//
refGorn.xPowerOnFeedback:=xPowerOnFeedback;
refGorn.xInterlock:=xInterlock;
refGorn.xPowerEnable:= refGornRegisters.Read.strPowerSupplyControlRegister.sValue.COIL_VALUE[0];

{region "Blocked"}
IF refGorn.xInterlock  THEN
	refGorn.xBlocked:=TRUE;
ELSE
	refGorn.xBlocked:=FALSE;
END_IF
{endregion}
	 
{region "Setpoint check"}
refGorn.xAutoMode:=refGornSetting.xAutoMode;
refGorn.xModbusConnected:=xModbusConnected;	 
IF refGornSetting.xAutoMode THEN	 
	SpCurrent:=LIMIT(refGornSetting.rMinSpCurrent,refGornSetting.rAutoModeCurrent , refGornSetting.rMaxSpCurrent);
ELSE
	SpCurrent:=LIMIT(refGornSetting.rMinSpCurrent,refGornSetting.rSpCurrent , refGornSetting.rMaxSpCurrent); 
END_IF;
SpVoltage:=LIMIT(refGornSetting.rMinSpVoltage, refGornSetting.rSpVoltage , refGornSetting.rMaxSpVoltage);
{endregion}

refGorn.rSpCurrentFeedback :=refGornRegisters.Read.strSpCurrent.sValue.INT_VALUE;
										

refGorn.rSpVoltageFeedback := refGornRegisters.Read.strSpVoltage.sValue.INT_VALUE;
IF xCommand AND refGorn.xPowerEnable THEN
	refGorn.rFbCurrent := refGornRegisters.Read.strFbCurrent.sValue.INT_VALUE;
								
	refGorn.rFbVoltage := refGornRegisters.Read.strFbVolatge.sValue.INT_VALUE;						
ELSE
	refGorn.rFbCurrent := 0 ;
	refGorn.rFbVoltage := 0;
END_IF
{endregion}
	 
{region "Command"}
IF refGornSetting.xAutoMode AND NOT refGorn.xBlocked THEN
		refGorn.xManualCommand:=refGorn.xAutoCommand;
		refGorn.xManualPowerCommand:=refGorn.xAutoPowerCommand;
		
			
		xCommand:=refgorn.xAutoCommand;	 
END_IF
	 
IF NOT refGornSetting.xAutoMode AND NOT refGorn.xBlocked THEN
		refGorn.xAutoCommand:=refGorn.xManualCommand;
		refGorn.xAutoPowerCommand:=refGorn.xManualPowerCommand;
		
		xCommand:=refgorn.xManualCommand;	 
END_IF
	//OR refGorn.xStabVoltageError
IF  refGorn.xInternalError  OR refGorn.xStabCurrentError OR refGorn.xPowerError OR refGorn.xHeatProtect THEN
	refGorn.xAutoCommand:=			FALSE;
	
	refGorn.xManualCommand:= 		FALSE;


	xCommand:=						FALSE;
	refGorn.xError:=				TRUE;
	 
END_IF

IF refGorn.xBlocked THEN
	refGorn.xAutoCommand:=			FALSE;
	
	refGorn.xManualCommand:= 		FALSE;


	xCommand:=						FALSE;
END_IF
{endregion}

{region "CommandCoil"}

refGornRegisters.Write.strPowerSupplyControlRegister.sValue.COIL_VALUE[0]:=refGorn.xAutoPowerCommand OR refGorn.xManualPowerCommand ;
refGornRegisters.Write.strPowerSupplyControlRegister.sValue.COIL_VALUE[1]:=xCommand;
{endregion}
refGornRegisters.Write.strSpCurrent.sValue.INT_VALUE:=SpCurrent;
refGornRegisters.Write.strSpVoltage.sValue.INT_VALUE:=SpVoltage;	 
{region "ErrorStatus"}
IF refGornRegisters.Read.strPowerSupplyStatusRegister.sValue.COIL_VALUE[0] THEN
	refGorn.xInternalError:=TRUE;	 
END_IF
IF refGornRegisters.Read.strPowerSupplyStatusRegister.sValue.COIL_VALUE[1] THEN
	refGorn.xStabVoltageError:=TRUE;		 
END_IF
IF refGornRegisters.Read.strPowerSupplyStatusRegister.sValue.COIL_VALUE[2] THEN
	refGorn.xStabCurrentError:=TRUE;	 
END_IF
IF refGornRegisters.Read.strPowerSupplyStatusRegister.sValue.COIL_VALUE[3] THEN
	refGorn.xPowerError:= TRUE;	 
END_IF
IF refGornRegisters.Read.strPowerSupplyStatusRegister.sValue.COIL_VALUE[4] THEN
	refGorn.xHeatProtect:=TRUE;	 
END_IF
	 

IF xCommand AND refGorn.xPowerEnable AND refGorn.rFbCurrent>0.0 AND refGorn.rFbVoltage>0.0 THEN
	refGorn.xTurnOn:=TRUE;
ELSE
	refGorn.xTurnOn:=FALSE;		 
END_IF
		  
			   
IF refGorn.xAcknowledge THEN
	refGorn.xAcknowledge:=FALSE;
	refGorn.xInternalError:=FALSE;
 	refGorn.xStabVoltageError:=FALSE;
	refGorn.xStabCurrentError:=FALSE;
	refGorn.xPowerError:= FALSE;
	refGorn.xHeatProtect:=FALSE;		
	refGorn.xError:=FALSE; 
END_IF
{endregion}


	 


{region "output"}
xInternalError:=refGorn.xInternalError;
xStabVoltageError:=refGorn.xStabVoltageError;
xStabCurrentError:=refGorn.xStabCurrentError;
xPowerError:=refGorn.xPowerError;
xHeatProtect:=refGorn.xHeatProtect;
xRemoteStatus:=refGorn.xRemoteStatus;
xError:=refGorn.xError;
{endregion}

END_FUNCTION_BLOCK

// Function Blocks/Heater/fbHeater
FUNCTION_BLOCK fbHeater
VAR_INPUT
	Heater: 	REFERENCE TO udtHeater;
	Setting:	REFERENCE TO udtHeaterSetting;
	xInterlock:	BOOL;
	Temperature: REAL;
	TransIsOn:BOOL;
END_VAR
VAR_OUTPUT
	Power: UDINT;
	Command:BOOL;
END_VAR
VAR
	Regulator: Util.PID;
	LimitsActive:BOOL;
	Overflow:BOOL;
	SetPoint: REAL:=0;
END_VAR

Setting.rManualPower:=LIMIT(Setting.rMinPower, Setting.rManualPower, Setting.rMaxPower);
Heater.xPowerOn:=TransIsOn;
Heater.xLock := xInterlock;
Heater.Temepature:=THIS^.Temperature;

Heater.xError:= NOT Heater.xPowerOn OR Overflow;
SetPoint:=Setting.rSetpointTemperature;

IF Heater.xError OR Heater.xLock THEN
	SetPoint:=0;
	Heater.xManualCommand:=FALSE;
	Heater.xAutoCommand:=FALSE;
	
END_IF
IF  NOT Heater.xCommand THEN
	SetPoint:=0;
END_IF

Regulator(	ACTUAL:=Heater.Temepature,
			SET_POINT:=SetPoint,
			KP:= Setting.P,
			TN:= Setting.I,
			TV:= Setting.D,
			Y_Manual:=Setting.rManualPower*100,
			Y_OFFSET:=0,
			Y_MIN:=0.0,
			Y_MAX:=Setting.rMaxPower*100,
			MANUAL:= Setting.xManualPower,
			RESET:=Heater.xReset,
			Y=>Heater.rPower,
			LIMITS_ACTIVE=>LimitsActive,
			OVERFLOW=>Overflow);


	
IF NOT Setting.xAutoMode THEN
	Heater.xCommand:=Heater.xManualCommand;
	Heater.xAutoCommand:=Heater.xManualCommand;
ELSE
	Heater.xCommand:=Heater.xAutoCommand;
	Heater.xManualCommand:=Heater.xAutoCommand;
END_IF
 
IF Heater.xError THEN
	Heater.wState:=2;
ELSIF Heater.xLock THEN
	Heater.wState:=3;
ELSIF Heater.xCommand THEN
	Heater.wState:=1;
ELSE
	Heater.wState:=0;
END_IF

Command:=Heater.xCommand;
Power:=REAL_TO_UDINT(Heater.rPower);

END_FUNCTION_BLOCK

// Function Blocks/Inficon/fbInficon
FUNCTION_BLOCK fbInficon
VAR_INPUT
	Inficon:			REFERENCE TO udtInficon;
	SendSize:  			REFERENCE TO UINT;
	pSendBuffer:		POINTER TO BYTE; //Указатель на массив отправки сообщения
	iSendBufferLength: 	INT;
	pRcvBuffer:			POINTER TO BYTE;
	pRcvSize:			INT; //Количество полученных байт;
	xSendMessageReady:	REFERENCE TO BOOL;//Сигнал о готовности сообщения для отправки
	xRcvFlagDone:		BOOL; //Флаг о завершение принятия данных
	pMessageBuffer: 	POINTER TO BYTE; //Указатель на байтовый массив, который будет использоваться как буффер для составления Message
	iMessageBuffferLength: INT;//Длина массива, который используется как буффер
	COMPortIsOpened:	BOOL;
	
	InficonResponce: POINTER TO udtInficonResponcePackage;
	
	InficonRemoteGeneralActionResponce: POINTER TO udtRemoteGeneralActionResponce;
END_VAR
VAR_OUTPUT
END_VAR
VAR
	MessageBuffer:		fbGeneralBuffer;//Функциональный блок для работы с буффером
	SendBuffer:			fbGeneralBuffer;
	
	Query: 				fbInficonQuery;
	Update: 			fbInficonUpdate;
	Status:				fbInficonStatus;
	Remote:				fbInficonRemote;
	STAGE: 				INT;
	xMesaageBufferEmpty:BOOL;
	xMessageBufferInit: BOOL:=FALSE;
	xSendBufferEmpty:	BOOL;
	HelloComadResult: 	INT;

	RawMessageLength: 	DINT;
	BufferPointer: 		POINTER TO ARRAY[0..1] OF BYTE;
	
	SensoreStatusResult:INT; //Реультат выполнения стадии опроса сенсоров
	CRCResult: 			BYTE;
	
	SensoreStatusStage: INT; //Этапы выполнения стадии опроса сенсоров
	RemoteGeneralActionResult: 	INT; //Результат выполнения стадии команд
	RemoteGeneralActionStage:	INT;
	
	getFiltredRateStage: INT;
	getFiltredRateRsult: INT;
	InficonResponceSMFilteredRate: udtInficonResponceSMFiltredrate;
	
	
	
END_VAR

IF NOT xMessageBufferInit THEN
	MessageBuffer(pBuffer:=pMessageBuffer,
			pBufferLength:=iMessageBuffferLength,
			xEmpty=>xMesaageBufferEmpty,
			xInit=>xMessageBufferInit);
	SendBuffer(	pBuffer:=pSendBuffer,
				pBufferLength:=iSendBufferLength,
				xEmpty=>xSendBufferEmpty,
				xInit=>xMessageBufferInit);
	THIS^.Status(MessageBuffer:=ADR(MessageBuffer));
	THIS^.Remote(MessageBuffer:=ADR(MessageBuffer));
	BufferPointer:=ADR(RawMessageLength);		
END_IF




CASE STAGE OF
	InficonStage.WAIT:
		IF COMPortIsOpened THEN
			STAGE:=InficonStage.STATUS_SENSORE;
		END_IF
		
	InficonStage.STATUS_SENSORE:
		SensoreStatusResult:=THIS^.SensoreStatus(SensoreStatusStage);
		IF SensoreStatusResult = InficonMethodStatus.COMPLETE THEN
			Stage:=InficonStage.GET_MATERIAL_FILTRED_RATE;
		END_IF
		IF SensoreStatusResult = InficonMethodStatus.ERROR THEN
			Stage:= InficonStage.ERROR;
		END_IF
	InficonStage.GET_MATERIAL_FILTRED_RATE:
		getFiltredRateRsult :=THIS^.GetMateriaFiltredRate(Stage:=getFiltredRateStage);
		IF getFiltredRateRsult = InficonMethodStatus.COMPLETE THEN
			Stage:=InficonStage.REMOTE_GENERAL_ACTION;
		END_IF
		IF getFiltredRateRsult = InficonMethodStatus.ERROR THEN
			Stage:= InficonStage.ERROR;
		END_IF		
	InficonStage.REMOTE_GENERAL_ACTION:
		IF Inficon.xManualReset_1 THEN
			RemoteGeneralActionResult:=THIS^.RemoteGeneralAction(RemoteGeneralActionStage,16#01);
			IF RemoteGeneralActionResult = InficonMethodStatus.COMPLETE THEN
				Inficon.xManualReset_1:=FALSE;
				Stage:=InficonStage.WAIT;
			END_IF
			IF RemoteGeneralActionResult = InficonMethodStatus.ERROR THEN
				Stage:= InficonStage.ERROR;
			END_IF
		ELSIF Inficon.xManualReset_2 THEN
			RemoteGeneralActionResult:=THIS^.RemoteGeneralAction(RemoteGeneralActionStage,16#02);
			IF RemoteGeneralActionResult = InficonMethodStatus.COMPLETE THEN
				Inficon.xManualReset_2:=FALSE;
				Stage:=InficonStage.WAIT;
			END_IF
			IF RemoteGeneralActionResult = InficonMethodStatus.ERROR THEN
				Stage:= InficonStage.ERROR;
			END_IF
		ELSIF Inficon.xManualReset_3 THEN
			RemoteGeneralActionResult:=THIS^.RemoteGeneralAction(RemoteGeneralActionStage,16#03);
			IF RemoteGeneralActionResult = InficonMethodStatus.COMPLETE THEN
				Inficon.xManualReset_3:=FALSE;
				Stage:=InficonStage.WAIT;
			END_IF
			IF RemoteGeneralActionResult = InficonMethodStatus.ERROR THEN
				Stage:= InficonStage.ERROR;
			END_IF
		ELSIF
			Inficon.xManualReset_4 THEN
			RemoteGeneralActionResult:=THIS^.RemoteGeneralAction(RemoteGeneralActionStage,16#04);
			IF RemoteGeneralActionResult = InficonMethodStatus.COMPLETE THEN
				Inficon.xManualReset_4:=FALSE;
				Stage:=InficonStage.WAIT;
			END_IF
			IF RemoteGeneralActionResult = InficonMethodStatus.ERROR THEN
				Stage:= InficonStage.ERROR;
			END_IF
		ELSIF Inficon.xManualReset_5 THEN
			RemoteGeneralActionResult:=THIS^.RemoteGeneralAction(RemoteGeneralActionStage,16#05);
			IF RemoteGeneralActionResult = InficonMethodStatus.COMPLETE THEN
				Inficon.xManualReset_5:=FALSE;
				Stage:=InficonStage.WAIT;
			END_IF
			IF RemoteGeneralActionResult = InficonMethodStatus.ERROR THEN
				Stage:= InficonStage.ERROR;
			END_IF
		ELSIF Inficon.xManualReset_6 THEN
			RemoteGeneralActionResult:=THIS^.RemoteGeneralAction(RemoteGeneralActionStage,16#06);
			IF RemoteGeneralActionResult = InficonMethodStatus.COMPLETE THEN
				Inficon.xManualReset_6:=FALSE;
				Stage:=InficonStage.WAIT;
			END_IF
			IF RemoteGeneralActionResult = InficonMethodStatus.ERROR THEN
				Stage:= InficonStage.ERROR;
			END_IF
		ELSE
			Stage:=InficonStage.WAIT;
		END_IF
		

	InficonStage.ERROR:
		IF Inficon.xAcknowledge THEN
			Inficon.xAcknowledge:=FALSE;
			Stage:=InficonStage.WAIT;
		END_IF
	
// 	
// 	10:
// 		HelloComadResult:=THIS^.HelloCommand(16#01);
// 		IF HelloComadResult<>-1 THEN
// 			Stage:=11;
// 		END_IF
// 	11:
// 		RawMessageLength:=MessageBuffer.getBufferLength;
// 
// 		SendBuffer.AddElement(BufferPointer^[0]);
// 		SendBuffer.AddElement(BufferPointer^[1]);
// 		Stage:=12;
// 	12:
// 		SendBuffer.AddStruct(pData:=MessageBuffer.getBufferAddres,
// 							Length:=DINT_TO_INT(MessageBuffer.getBufferLength));
// 		Stage:=13;
// 	13:
// 		CRCResult:=THIS^.CalcCRC(Message:=SendBuffer.getBufferAddres,
// 									Length:=SendBuffer.getBufferLength);
// 		Stage:=14;
// 	14:
// 		SendBuffer.AddElement(THIS^.CRCResult);
// 		xSendMessageReady:=TRUE;
// 		Stage:=0;
// 		
		
END_CASE

METHOD ADD_Sensore : INT
VAR_INPUT
	SensoreNumber: BYTE;
END_VAR
END_METHOD

(*Расчет CRC*)
METHOD CalcCRC : BYTE
VAR_INPUT
	Message: POINTER TO BYTE;
	Length: DINT;
END_VAR
VAR
	Counter: DINT;
	InnerMessage: POINTER TO BYTE;
END_VAR
CalcCRC:=0;

FOR Counter:=0 TO Length-1 DO
	InnerMessage :=Message+Counter;
	CalcCRC:=CalcCRC+InnerMessage^;
END_FOR

CalcCRC:=CalcCRC AND 255;
END_METHOD

METHOD GetMateriaFiltredRate : INT
VAR_INPUT
	Stage: 					REFERENCE TO INT;
END_VAR
VAR
	AddCommandResult: 		INT;
	ClearMessageResult: 	INT; //Результат выполнения отчистки буффера сообщений
	ClearSendBufferResult:	INT; //Результат выполнения очистки буффера отправки
	RawLength: 				DINT;
	MessageLengthForBuffer: POINTER TO ARRAY[0..1] OF BYTE;
	CRCResult: 				BYTE;
	rTempFloat:				POINTER TO REAL;
END_VAR
CASE Stage OF
	InficonMethodStage.WAIT:
		GetMateriaFiltredRate:=InficonMethodState.BUSY;
		ClearMessageResult:=THIS^.MessageBuffer.ClearBuffer();
		ClearSendBufferResult:=THIS^.SendBuffer.ClearBuffer();
		IF ClearMessageResult = 200 AND ClearSendBufferResult = 200 THEN
			Stage:=InficonMethodStage.ADD_COMMAND;
		END_IF
	InficonMethodStage.ADD_COMMAND:
		AddCommandResult:=THIS^.Status.Material(CommandID:=InficonSLCommandID.FilteredRate, MaterialNumber:=16#0);
		IF AddCommandResult = -1THEN
			GetMateriaFiltredRate := InficonMethodState.ERROR;
			RETURN;
		END_IF
		Stage:=InficonMethodStage.ADD_LENGTH_TO_SENDBUFFER;
	InficonMethodStage.ADD_LENGTH_TO_SENDBUFFER:
		RawLength:=THIS^.MessageBuffer.getBufferLength;
		MessageLengthForBuffer:=ADR(RawLength);
		THIS^.SendBuffer.AddElement(pData:=MessageLengthForBuffer^[0]);
		THIS^.SendBuffer.AddElement(pData:=MessageLengthForBuffer^[1]);
		Stage:=InficonMethodStage.CALC_CRC;
	InficonMethodStage.CALC_CRC:
		CRCResult:=THIS^.CalcCRC(Message:=THIS^.MessageBuffer.getBufferAddres,
									Length:=THIS^.MessageBuffer.getBufferLength);
		THIS^.MessageBuffer.AddElement(pData:=CRCResult);
		Stage:=InficonMethodStage.ADD_CRC;
	InficonMethodStage.ADD_CRC:
		Stage:=InficonMethodStage.ADD_DATA_TO_SENDBUFFER;
	InficonMethodStage.ADD_DATA_TO_SENDBUFFER:
		THIS^.SendBuffer.AddStruct(pData:=THIS^.MessageBuffer.getBufferAddres,
								Length:=DINT_TO_INT(THIS^.MessageBuffer.getBufferLength));
		Stage:=InficonMethodStage.EDGE_MESSAGECOMPLETE_FLAG;		
	InficonMethodStage.EDGE_MESSAGECOMPLETE_FLAG:
		THIS^.SendSize:=DINT_TO_UINT(THIS^.SendBuffer.getBufferLength);
		THIS^.xSendMessageReady:=TRUE;
		Stage:=InficonMethodStage.WAIT_RESPONCE;
	InficonMethodStage.WAIT_RESPONCE:
		IF THIS^.xRcvFlagDone THEN
			Stage:=InficonMethodStage.PARSE_RESPONCE;
		END_IF
	InficonMethodStage.PARSE_RESPONCE:
		MEMUtils.MemCpy(pbyDest:=ADR(THIS^.InficonResponceSMFilteredRate),
						pbySrc:=pRcvBuffer,
						dwSize:=5);
		Stage:=InficonMethodStage.CHECK_RESPONCE_STATUS;		
	InficonMethodStage.CHECK_RESPONCE_STATUS:
		IF InficonResponceSMFilteredRate.Code<>16#6 THEN
			Stage:=InficonMethodStage.COMPLETE;
			RETURN;
		END_IF
		
		MEMUtils.MemCpy(pbyDest:=ADR(THIS^.InficonResponceSMFilteredRate),
						pbySrc:=pRcvBuffer,
						dwSize:=SIZEOF(udtInficonResponceSMFiltredrate));
						
		THIS^.Inficon.Materials.FilteredRate[0].vValue[0]:=InficonResponceSMFilteredRate.FR_1_1;
		THIS^.Inficon.Materials.FilteredRate[0].vValue[1]:=InficonResponceSMFilteredRate.FR_1_2;
		THIS^.Inficon.Materials.FilteredRate[0].vValue[2]:=InficonResponceSMFilteredRate.FR_1_3;
		THIS^.Inficon.Materials.FilteredRate[0].vValue[3]:=InficonResponceSMFilteredRate.FR_1_4;

		THIS^.Inficon.Materials.FilteredRate[1].vValue[0]:=InficonResponceSMFilteredRate.FR_2_1;
		THIS^.Inficon.Materials.FilteredRate[1].vValue[1]:=InficonResponceSMFilteredRate.FR_2_2;
		THIS^.Inficon.Materials.FilteredRate[1].vValue[2]:=InficonResponceSMFilteredRate.FR_2_3;
		THIS^.Inficon.Materials.FilteredRate[1].vValue[3]:=InficonResponceSMFilteredRate.FR_2_4;
		
		THIS^.Inficon.Materials.FilteredRate[2].vValue[0]:=InficonResponceSMFilteredRate.FR_3_1;
		THIS^.Inficon.Materials.FilteredRate[2].vValue[1]:=InficonResponceSMFilteredRate.FR_3_2;
		THIS^.Inficon.Materials.FilteredRate[2].vValue[2]:=InficonResponceSMFilteredRate.FR_3_3;
		THIS^.Inficon.Materials.FilteredRate[2].vValue[3]:=InficonResponceSMFilteredRate.FR_3_4;

		THIS^.Inficon.Materials.FilteredRate[3].vValue[0]:=InficonResponceSMFilteredRate.FR_4_1;
		THIS^.Inficon.Materials.FilteredRate[3].vValue[1]:=InficonResponceSMFilteredRate.FR_4_2;
		THIS^.Inficon.Materials.FilteredRate[3].vValue[2]:=InficonResponceSMFilteredRate.FR_4_3;
		THIS^.Inficon.Materials.FilteredRate[3].vValue[3]:=InficonResponceSMFilteredRate.FR_4_4;

		THIS^.Inficon.Materials.FilteredRate[4].vValue[0]:=InficonResponceSMFilteredRate.FR_5_1;
		THIS^.Inficon.Materials.FilteredRate[4].vValue[1]:=InficonResponceSMFilteredRate.FR_5_2;
		THIS^.Inficon.Materials.FilteredRate[4].vValue[2]:=InficonResponceSMFilteredRate.FR_5_3;
		THIS^.Inficon.Materials.FilteredRate[4].vValue[3]:=InficonResponceSMFilteredRate.FR_5_4;

		THIS^.Inficon.Materials.FilteredRate[5].vValue[0]:=InficonResponceSMFilteredRate.FR_6_1;
		THIS^.Inficon.Materials.FilteredRate[5].vValue[1]:=InficonResponceSMFilteredRate.FR_6_2;
		THIS^.Inficon.Materials.FilteredRate[5].vValue[2]:=InficonResponceSMFilteredRate.FR_6_3;
		THIS^.Inficon.Materials.FilteredRate[5].vValue[3]:=InficonResponceSMFilteredRate.FR_6_4;
		
		Stage:=InficonMethodStage.COMPLETE;
	InficonMethodStage.COMPLETE:
		Stage:=InficonMethodStage.WAIT;
		GetMateriaFiltredRate:=InficonMethodStatus.COMPLETE;
	InficonMethodStage.ERROR:
	
	
	
END_CASE
END_METHOD

METHOD HCPub : INT
VAR_INPUT
	CommandID:BYTE;
END_VAR
HCPub:=HelloCommand(CommandID:=CommandID);
END_METHOD

(*
HelloComand - метод формируюзий Hello Command запрос
Формат запроса: H<CommandID>
*)
METHOD PROTECTED HelloCommand : INT
VAR_INPUT
	CommandID:BYTE;
END_VAR
VAR
	CRC:BYTE;
END_VAR
THIS^.MessageBuffer.ClearBuffer();
HelloCommand:=THIS^.MessageBuffer.AddElement(pData:=InficonCommand.Hello,
							);
IF HelloCommand = -1 THEN
	RETURN;
END_IF
	
HelloCommand:=THIS^.MessageBuffer.AddElement(pData:=CommandID,
							);

			
IF HelloCommand = -1 THEN
	RETURN;
END_IF
END_METHOD

METHOD RemoteGeneralAction : INT
VAR_INPUT
	Stage: REFERENCE TO INT;
	MaterialNumber: BYTE;
	
END_VAR
VAR
	ClearMessageResult: 	INT; //Результат выполнения отчистки буффера сообщений
	ClearSendBufferResult:	INT; //Результат выполнения очистки буффера отправки
	AddCommandResult: 		INT;
	RawLength: 				DINT; //Длина сообщения
	MessageLengthForBuffer: POINTER TO ARRAY[0..1] OF BYTE;
	CRCResult: 				BYTE; 
	
	
END_VAR
CASE Stage OF
	

	InficonMethodStage.WAIT:
		RemoteGeneralAction:=InficonMethodState.BUSY;
		ClearMessageResult:=THIS^.MessageBuffer.ClearBuffer();
		ClearSendBufferResult:=THIS^.SendBuffer.ClearBuffer();
		IF ClearMessageResult = 200 AND ClearSendBufferResult = 200 THEN
			Stage:=InficonMethodStage.ADD_COMMAND;
		END_IF
	
		
	InficonMethodStage.ADD_COMMAND:
		AddCommandResult:=THIS^.Remote.MaterialAction(CommandID:=InficonRLCommandID.ZeroThickness,
													MaterialNumber:=MaterialNumber,
													pData:=0,
													Length:=0);
		IF AddCommandResult= -1 THEN
			RemoteGeneralAction:=InficonMethodState.ERROR;
			RETURN;
		END_IF
		Stage:=InficonMethodStage.ADD_LENGTH_TO_SENDBUFFER;
	
		
	InficonMethodStage.ADD_LENGTH_TO_SENDBUFFER:
		RawLength:=THIS^.MessageBuffer.getBufferLength;
		MessageLengthForBuffer:=ADR(RawLength);
		THIS^.SendBuffer.AddElement(pData:=MessageLengthForBuffer^[0]);
		THIS^.SendBuffer.AddElement(pData:=MessageLengthForBuffer^[1]);
		Stage:=InficonMethodStage.CALC_CRC;
		
		
	InficonMethodStage.CALC_CRC:
		CRCResult:=THIS^.CalcCRC(Message:=THIS^.MessageBuffer.getBufferAddres,
									Length:=THIS^.MessageBuffer.getBufferLength);
		THIS^.MessageBuffer.AddElement(pData:=CRCResult);
		Stage:=InficonMethodStage.ADD_DATA_TO_SENDBUFFER;
		
		
	InficonMethodStage.ADD_DATA_TO_SENDBUFFER:
		THIS^.SendBuffer.AddStruct(pData:=THIS^.MessageBuffer.getBufferAddres,
								Length:=DINT_TO_INT(THIS^.MessageBuffer.getBufferLength));
		Stage:=InficonMethodStage.EDGE_MESSAGECOMPLETE_FLAG;
		
		
	InficonMethodStage.EDGE_MESSAGECOMPLETE_FLAG:
		THIS^.SendSize:=DINT_TO_UINT(THIS^.SendBuffer.getBufferLength);
		THIS^.xSendMessageReady:=TRUE;
		Stage:=InficonMethodStage.WAIT_RESPONCE;
	
		
	InficonMethodStage.WAIT_RESPONCE:
		IF THIS^.xRcvFlagDone THEN
			Stage:=InficonMethodStage.PARSE_RESPONCE;
		END_IF
	
		
	InficonMethodStage.PARSE_RESPONCE:
		MEMUtils.MemCpy(pbyDest:=THIS^.InficonRemoteGeneralActionResponce,
						pbySrc:=pRcvBuffer,
						dwSize:=THIS^.pRcvSize);
		Stage:=InficonMethodStage.CHECK_RESPONCE_STATUS;
	
		
	InficonMethodStage.CHECK_RESPONCE_STATUS:
	
			Stage:=InficonMethodStage.COMPLETE;

		THIS^.xSendMessageReady:=FALSE;
		THIS^.xRcvFlagDone:=TRUE;
		
		
	InficonMethodStage.COMPLETE:
		Stage:=InficonMethodStage.WAIT;
		RemoteGeneralAction:=InficonMethodStatus.COMPLETE;
		
	InficonMethodStage.ERROR:
END_CASE
END_METHOD

METHOD SensoreStatus : INT
VAR_INPUT
	Stage: REFERENCE TO INT;
END_VAR
VAR
	AddCommandResult: INT;
	ClearMessageResult: INT; //Результат выполнения отчистки буффера сообщений
	ClearSendBufferResult:INT; //Результат выполнения очистки буффера отправки
	RawLength: DINT;
	MessageLengthForBuffer: POINTER TO ARRAY[0..1] OF BYTE;
	CRCResult: BYTE;
	rTempFloat:POINTER TO REAL;
	
END_VAR
CASE Stage OF
	InficonMethodStage.WAIT:
	
		//Инициализация массивов
		SensoreStatus:=InficonMethodState.BUSY;
		ClearMessageResult:=THIS^.MessageBuffer.ClearBuffer();
		ClearSendBufferResult:=THIS^.SendBuffer.ClearBuffer();
		IF ClearMessageResult = 200 AND ClearSendBufferResult = 200 THEN
			Stage:=InficonMethodStage.ADD_COMMAND;
		END_IF
		
	InficonMethodStage.ADD_COMMAND:
		//Запись команды получения значения всех скоростей напыления
		AddCommandResult:=THIS^.Status.Sensor(CommandID:=InficonSSCommandID.SensorThickness, SensorNumber:=16#0);
		IF AddCommandResult= -1 THEN
			SensoreStatus:=InficonMethodState.ERROR;
			RETURN;
		END_IF
		Stage:=InficonMethodStage.ADD_LENGTH_TO_SENDBUFFER;

	InficonMethodStage.ADD_LENGTH_TO_SENDBUFFER:
	
		RawLength:=THIS^.MessageBuffer.getBufferLength;
		MessageLengthForBuffer:=ADR(RawLength);
		THIS^.SendBuffer.AddElement(pData:=MessageLengthForBuffer^[0]);
		THIS^.SendBuffer.AddElement(pData:=MessageLengthForBuffer^[1]);
		Stage:=InficonMethodStage.CALC_CRC;
	
	InficonMethodStage.CALC_CRC:
		
		CRCResult:=THIS^.CalcCRC(Message:=THIS^.MessageBuffer.getBufferAddres,
									Length:=THIS^.MessageBuffer.getBufferLength);
		THIS^.MessageBuffer.AddElement(pData:=CRCResult);
		Stage:=InficonMethodStage.ADD_CRC;
		
	InficonMethodStage.ADD_CRC:
		Stage:=InficonMethodStage.ADD_DATA_TO_SENDBUFFER;
		
	InficonMethodStage.ADD_DATA_TO_SENDBUFFER:
		THIS^.SendBuffer.AddStruct(pData:=THIS^.MessageBuffer.getBufferAddres,
								Length:=DINT_TO_INT(THIS^.MessageBuffer.getBufferLength));
		Stage:=InficonMethodStage.EDGE_MESSAGECOMPLETE_FLAG;
		
	InficonMethodStage.EDGE_MESSAGECOMPLETE_FLAG:
		THIS^.SendSize:=DINT_TO_UINT(THIS^.SendBuffer.getBufferLength);
		THIS^.xSendMessageReady:=TRUE;
		Stage:=InficonMethodStage.WAIT_RESPONCE;
		
	InficonMethodStage.WAIT_RESPONCE:
		IF THIS^.xRcvFlagDone THEN
			Stage:=InficonMethodStage.PARSE_RESPONCE;
		END_IF
	InficonMethodStage.PARSE_RESPONCE:
		MEMUtils.MemCpy(pbyDest:=InficonResponce,
						pbySrc:=pRcvBuffer,
						dwSize:=5);
		Stage:=InficonMethodStage.CHECK_RESPONCE_STATUS;
		
	InficonMethodStage.CHECK_RESPONCE_STATUS:
		IF InficonResponce^.Code<>16#6 THEN
			Stage:=InficonMethodStage.COMPLETE;
			RETURN;
		END_IF
		
		MEMUtils.MemCpy(pbyDest:=InficonResponce,
						pbySrc:=pRcvBuffer,
						dwSize:=SIZEOF(udtInficonResponcePackage));
						
		(*MEMUtils.SwapLocalToMotorola(pAddress:=ADR(InficonResponce^.Thinkness_1_1),
								iSize:=4);
		rTempFloat:= ADR(InficonResponce^.Thinkness_1_1);
		THIS^.Inficon.Sensore1Thickness:=rTempFloat^;*)
		THIS^.Inficon.Sensore1Thickness.vValue[0]:=InficonResponce^.Thinkness_1_1;
		THIS^.Inficon.Sensore1Thickness.vValue[1]:=InficonResponce^.Thinkness_1_2;
		THIS^.Inficon.Sensore1Thickness.vValue[2]:=InficonResponce^.Thinkness_1_3;
		THIS^.Inficon.Sensore1Thickness.vValue[3]:=InficonResponce^.Thinkness_1_4;

		THIS^.Inficon.Sensore2Thickness.vValue[0]:=InficonResponce^.Thinkness_2_1;
		THIS^.Inficon.Sensore2Thickness.vValue[1]:=InficonResponce^.Thinkness_2_2;
		THIS^.Inficon.Sensore2Thickness.vValue[2]:=InficonResponce^.Thinkness_2_3;
		THIS^.Inficon.Sensore2Thickness.vValue[3]:=InficonResponce^.Thinkness_2_4;
		
		THIS^.Inficon.Sensore3Thickness.vValue[0]:=InficonResponce^.Thinkness_3_1;
		THIS^.Inficon.Sensore3Thickness.vValue[1]:=InficonResponce^.Thinkness_3_2;
		THIS^.Inficon.Sensore3Thickness.vValue[2]:=InficonResponce^.Thinkness_3_3;
		THIS^.Inficon.Sensore3Thickness.vValue[3]:=InficonResponce^.Thinkness_3_4;

		THIS^.Inficon.Sensore4Thickness.vValue[0]:=InficonResponce^.Thinkness_4_1;
		THIS^.Inficon.Sensore4Thickness.vValue[1]:=InficonResponce^.Thinkness_4_2;
		THIS^.Inficon.Sensore4Thickness.vValue[2]:=InficonResponce^.Thinkness_4_3;
		THIS^.Inficon.Sensore4Thickness.vValue[3]:=InficonResponce^.Thinkness_4_4;

		THIS^.Inficon.Sensore5Thickness.vValue[0]:=InficonResponce^.Thinkness_5_1;
		THIS^.Inficon.Sensore5Thickness.vValue[1]:=InficonResponce^.Thinkness_5_2;
		THIS^.Inficon.Sensore5Thickness.vValue[2]:=InficonResponce^.Thinkness_5_3;
		THIS^.Inficon.Sensore5Thickness.vValue[3]:=InficonResponce^.Thinkness_5_4;

		THIS^.Inficon.Sensore6Thickness.vValue[0]:=InficonResponce^.Thinkness_6_1;
		THIS^.Inficon.Sensore6Thickness.vValue[1]:=InficonResponce^.Thinkness_6_2;
		THIS^.Inficon.Sensore6Thickness.vValue[2]:=InficonResponce^.Thinkness_6_3;
		THIS^.Inficon.Sensore6Thickness.vValue[3]:=InficonResponce^.Thinkness_6_4;
		Stage:=InficonMethodStage.COMPLETE;
		
		
		
		
	InficonMethodStage.COMPLETE:
		Stage:=InficonMethodStage.WAIT;
		SensoreStatus:=InficonMethodStatus.COMPLETE;
	InficonMethodStage.ERROR:
END_CASE
END_METHOD

END_FUNCTION_BLOCK

// Function Blocks/Inficon/fbInficonQuery
FUNCTION_BLOCK fbInficonQuery
VAR_INPUT
	MessageBuffer: POINTER TO fbGeneralBuffer;
END_VAR
VAR_OUTPUT
END_VAR
VAR
END_VAR

THIS^.MessageBuffer^.ClearBuffer();
THIS^.MessageBuffer^.AddElement(pData:=InficonCommand.Query,);

(*
QG<CommandID>
*)
METHOD PUBLIC General : INT
VAR_INPUT
	CommandID:BYTE;
END_VAR
THIS^();

General:=THIS^.MessageBuffer^.AddElement(pData:=InficonQUSubgroup.General);
IF General = -1 THEN
	RETURN;
END_IF

General:=THIS^.MessageBuffer^.AddElement(pData:=CommandID);	
IF General = -1 THEN
	RETURN;
END_IF
END_METHOD

METHOD PUBLIC Material : INT
VAR_INPUT
	CommandID: BYTE;
	MaterialNumber:BYTE;
END_VAR
THIS^();

Material:= THIS^.MessageBuffer^.AddElement(pData:=InficonQUSubgroup.Material);
IF Material = -1 THEN
	RETURN;
END_IF

Material:= THIS^.MessageBuffer^.AddElement(pData:=CommandID);
IF Material = -1 THEN
	RETURN;
END_IF

Material:= THIS^.MessageBuffer^.AddElement(pData:=MaterialNumber);
IF Material = -1 THEN
	RETURN;
END_IF
END_METHOD

METHOD PUBLIC ProcessMaterial : INT
VAR_INPUT
	CommandID: BYTE;
	ProcessNumber:BYTE;
	MaterialNumber:BYTE;
END_VAR
THIS^();



ProcessMaterial:= THIS^.MessageBuffer^.AddElement(pData:=InficonQUSubgroup.Process);
IF ProcessMaterial = -1 THEN
	RETURN;
END_IF



ProcessMaterial:= THIS^.MessageBuffer^.AddElement(pData:=CommandID);
IF ProcessMaterial = -1 THEN
	RETURN;
END_IF

ProcessMaterial:= THIS^.MessageBuffer^.AddElement(pData:=ProcessNumber);
IF ProcessMaterial = -1 THEN
	RETURN;
END_IF

ProcessMaterial:= THIS^.MessageBuffer^.AddElement(pData:=MaterialNumber);
IF ProcessMaterial = -1 THEN
	RETURN;
END_IF
END_METHOD

METHOD PUBLIC Sensor : INT
VAR_INPUT
	CommandID: BYTE;
	SensorNumber:BYTE;
END_VAR
THIS^();

Sensor:= THIS^.MessageBuffer^.AddElement(pData:=InficonQUSubgroup.Sensor);
IF Sensor = -1 THEN
	RETURN;
END_IF

Sensor:= THIS^.MessageBuffer^.AddElement(pData:=CommandID);
IF Sensor = -1 THEN
	RETURN;
END_IF

Sensor:= THIS^.MessageBuffer^.AddElement(pData:=SensorNumber);
IF Sensor = -1 THEN
	RETURN;
END_IF
END_METHOD

METHOD PUBLIC Source : INT
VAR_INPUT	
	CommandID: BYTE;
	SourceNumber:BYTE;
END_VAR
THIS^();

Source:= THIS^.MessageBuffer^.AddElement(pData:=InficonQUSubgroup.Source);
IF Source = -1 THEN
	RETURN;
END_IF

Source:= THIS^.MessageBuffer^.AddElement(pData:=CommandID);
IF Source = -1 THEN
	RETURN;
END_IF

Source:= THIS^.MessageBuffer^.AddElement(pData:=SourceNumber);
IF Source = -1 THEN
	RETURN;
END_IF
END_METHOD

END_FUNCTION_BLOCK

// Function Blocks/Inficon/fbInficonUpdate
FUNCTION_BLOCK fbInficonUpdate
VAR_INPUT
	MessageBuffer: POINTER TO fbGeneralBuffer;
END_VAR
VAR_OUTPUT
END_VAR
VAR
END_VAR

THIS^.MessageBuffer^.ClearBuffer();
THIS^.MessageBuffer^.AddElement(pData:=InficonCommand.Update);

METHOD PUBLIC General : INT
VAR_INPUT
	CommandID:BYTE;
	pData: POINTER TO BYTE;
	Length:INT;
END_VAR
THIS^();

General := THIS^.MessageBuffer^.AddElement(pData:=InficonQUSubgroup.General);
IF General = -1 THEN
	RETURN;
END_IF

General:=THIS^.MessageBuffer^.AddElement(pData:=CommandID);
IF General= -1 THEN
	RETURN;
END_IF

General:=THIS^.MessageBuffer^.AddStruct(pData:=pData,
			Length:=Length);
IF General = -1 THEN
	RETURN;
END_IF
END_METHOD

METHOD PUBLIC Material : INT
VAR_INPUT
	CommandID: BYTE;
	MaterialNumber:BYTE;
	pData: POINTER TO BYTE;
	Length:INT;
END_VAR
THIS^();

Material:= THIS^.MessageBuffer^.AddElement(pData:=InficonQUSubgroup.Material);
IF Material = -1 THEN
	RETURN;
END_IF

Material:= THIS^.MessageBuffer^.AddElement(pData:=CommandID);
IF Material = -1 THEN
	RETURN;
END_IF

Material:= THIS^.MessageBuffer^.AddElement(pData:=MaterialNumber);
IF Material = -1 THEN
	RETURN;
END_IF

Material:=THIS^.MessageBuffer^.AddStruct(pData:=pData,
	Length:=Length);
IF Material = -1 THEN
	RETURN;
END_IF
END_METHOD

METHOD PUBLIC ProcessMaterial : INT
VAR_INPUT
	CommandID: BYTE;
	ProcessNumber:BYTE;
	MaterialNumber:BYTE;
	pData: POINTER TO BYTE;
	Length:INT;
END_VAR
THIS^();

ProcessMaterial:= THIS^.MessageBuffer^.AddElement(pData:=InficonQUSubgroup.Process);
IF ProcessMaterial = -1 THEN
	RETURN;
END_IF

ProcessMaterial:= THIS^.MessageBuffer^.AddElement(pData:=CommandID);
IF ProcessMaterial = -1 THEN
	RETURN;
END_IF

ProcessMaterial:= THIS^.MessageBuffer^.AddElement(pData:=ProcessNumber);
IF ProcessMaterial = -1 THEN
	RETURN;
END_IF

ProcessMaterial:= THIS^.MessageBuffer^.AddElement(pData:=MaterialNumber);
IF ProcessMaterial = -1 THEN
	RETURN;
END_IF

ProcessMaterial:=THIS^.MessageBuffer^.AddStruct(pData:=pData,
	Length:=Length);
IF ProcessMaterial = -1 THEN
	RETURN;
END_IF
END_METHOD

METHOD PUBLIC Sensor : INT
VAR_INPUT
	CommandID: BYTE;
	SensorNumber:BYTE;
	pData: POINTER TO BYTE;
	Length:INT;
END_VAR
THIS^();

Sensor:= THIS^.MessageBuffer^.AddElement(pData:=InficonQUSubgroup.Sensor);
IF Sensor = -1 THEN
	RETURN;
END_IF

Sensor:= THIS^.MessageBuffer^.AddElement(pData:=CommandID);
IF Sensor = -1 THEN
	RETURN;
END_IF

Sensor:= THIS^.MessageBuffer^.AddElement(pData:=SensorNumber);
IF Sensor = -1 THEN
	RETURN;
END_IF

Sensor:=THIS^.MessageBuffer^.AddStruct(pData:=pData,
	Length:=Length);
IF Sensor = -1 THEN
	RETURN;
END_IF
END_METHOD

METHOD PUBLIC Source : INT
VAR_INPUT
	CommandID: BYTE;
	SourceNumber:BYTE;
	pData: POINTER TO BYTE;
	Length:INT;
END_VAR
THIS^();

Source:= THIS^.MessageBuffer^.AddElement(pData:=InficonQUSubgroup.Sensor);
IF Source = -1 THEN
	RETURN;
END_IF

Source:= THIS^.MessageBuffer^.AddElement(pData:=CommandID);
IF Source = -1 THEN
	RETURN;
END_IF

Source:= THIS^.MessageBuffer^.AddElement(pData:=SourceNumber);
IF Source = -1 THEN
	RETURN;
END_IF

Source:=THIS^.MessageBuffer^.AddStruct(pData:=pData,
	Length:=Length);
IF Source = -1 THEN
	RETURN;
END_IF
END_METHOD

END_FUNCTION_BLOCK

// Function Blocks/Inficon/fbInficonStatus
FUNCTION_BLOCK fbInficonStatus
VAR_INPUT
	MessageBuffer: POINTER TO fbGeneralBuffer;
END_VAR
VAR_OUTPUT
END_VAR
VAR

END_VAR


THIS^.MessageBuffer^.AddElement(pData:=InficonCommand.Status);

METHOD PUBLIC Material : INT
VAR_INPUT
	CommandID: BYTE;
	MaterialNumber:BYTE;
END_VAR
THIS^();

Material:= THIS^.MessageBuffer^.AddElement(pData:=InficonRSSubgroup.Material);
IF Material = -1 THEN
	RETURN;
END_IF

Material:= THIS^.MessageBuffer^.AddElement(pData:=CommandID);
IF Material = -1 THEN
	RETURN;
END_IF

Material:= THIS^.MessageBuffer^.AddElement(pData:=MaterialNumber);
IF Material = -1 THEN
	RETURN;
END_IF
END_METHOD

METHOD PUBLIC Sensor : INT
VAR_INPUT
	CommandID: BYTE;
	SensorNumber:BYTE;
END_VAR
THIS^();

Sensor:= THIS^.MessageBuffer^.AddElement(pData:=InficonRSSubgroup.Sensor);
IF Sensor = -1 THEN
	RETURN;
END_IF

Sensor:= THIS^.MessageBuffer^.AddElement(pData:=CommandID);
IF Sensor = -1 THEN
	RETURN;
END_IF

Sensor:= THIS^.MessageBuffer^.AddElement(pData:=SensorNumber);
IF Sensor = -1 THEN
	RETURN;
END_IF
END_METHOD

END_FUNCTION_BLOCK

// Function Blocks/Inficon/fbInficonRemote
FUNCTION_BLOCK fbInficonRemote
VAR_INPUT
	MessageBuffer: POINTER TO fbGeneralBuffer;
END_VAR
VAR_OUTPUT
END_VAR
VAR
END_VAR

THIS^.MessageBuffer^.AddElement(pData:=InficonCommand.RemoteAction);

METHOD PUBLIC General : INT
VAR_INPUT
	CommandID:BYTE;
	pData: POINTER TO BYTE; //Pointer to ActionValue
	Length:INT;
END_VAR
THIS^();

General := THIS^.MessageBuffer^.AddElement(pData:=InficonRSSubgroup.General);
IF General = -1 THEN
	RETURN;
END_IF

General:=THIS^.MessageBuffer^.AddElement(pData:=CommandID);
IF General= -1 THEN
	RETURN;
END_IF

General:=THIS^.MessageBuffer^.AddStruct(pData:=pData,
			Length:=Length);
IF General = -1 THEN
	RETURN;
END_IF
END_METHOD

METHOD PUBLIC MaterialAction : INT
VAR_INPUT
	CommandID: BYTE;
	MaterialNumber:BYTE;
	pData: POINTER TO BYTE;
	Length:INT;
END_VAR
THIS^();

MaterialAction:= THIS^.MessageBuffer^.AddElement(pData:=InficonRSSubgroup.Material);
IF MaterialAction = -1 THEN
	RETURN;
END_IF

MaterialAction:= THIS^.MessageBuffer^.AddElement(pData:=CommandID);
IF MaterialAction = -1 THEN
	RETURN;
END_IF

MaterialAction:= THIS^.MessageBuffer^.AddElement(pData:=MaterialNumber);
IF MaterialAction = -1 THEN
	RETURN;
END_IF

IF pData <> 0 THEN
	MaterialAction:=THIS^.MessageBuffer^.AddStruct(pData:=pData,
			Length:=Length);
	IF MaterialAction = -1 THEN
		RETURN;
	END_IF
END_IF
END_METHOD

END_FUNCTION_BLOCK

// Function Blocks/IPS/IPSIon
FUNCTION_BLOCK IPSIon
VAR_INPUT
	refIPS:							REFERENCE TO udtIPS;
	Setting:						udtIPSSetting;
	xInterlock: 					BOOL;//Input: Внешняя блокировка
	xPowerOnFeedback:				BOOL;//Input: Обратная связь по питанию.
	rCurrentFeedback:				REAL;//Input: ОБратная связь по напряжению
	rVoltageFeedback:				REAL;//Input: Обратная связь по напряяжени.
	rPowerFeedback:					REAL;//Input: Обратная связь по мощности
	xTurnOn:						BOOL;//Input: Включен
	xError:							BOOL;//Input: ОШИБКА
	sStatus:						STRING;//Input: СТАТУС
	udtDeviceStatus:				REFERENCE TO unRegisterValue;
END_VAR
VAR_IN_OUT
	xStart:							BOOL;//OUTPUT:	Команда на старт 
	xStop:							BOOL;//OUTPUT: Команда на стоg
	xReset:							BOOL;//OUTPUT: Сброс ошибок
END_VAR


VAR
END_VAR

{region "input"}
refIPS.xInterlock:=xInterlock;
refIPS.xPowerOnFeedback:=xPowerOnFeedback;
refIPS.xTurnOn:=xTurnOn;
refIPS.xError:=xError;
refIPS.sStatus:=sStatus;
refIPS.rCurrentFeedback:=rCurrentFeedback;
refIPS.rVoltageFeedback:=rVoltageFeedback;
refIPS.rPowerFeedback:=rPowerFeedback;
{endregion}
	 
{region "Device Status"}
refIPS.xDeviceSwitchOn:=udtDeviceStatus.COIL_VALUE[0];
refIPS.xSmoothIncreseOutParametr:=udtDeviceStatus.COIL_VALUE[2];
refIPS.xSmoothDecreaseOutParametr:=udtDeviceStatus.COIL_VALUE[3];
refIPS.xInputConverterSwitchOn:=udtDeviceStatus.COIL_VALUE[4];
refIPS.xInputPowerOutOfLimit:=udtDeviceStatus.COIL_VALUE[5];
refIPS.xCriticalTemeratureWarning:=udtDeviceStatus.COIL_VALUE[6];
refIPS.xOverload:=udtDeviceStatus.COIL_VALUE[7];
refIPS.xOutPowerSitchingOn:=udtDeviceStatus.COIL_VALUE[8];
refIPS.xOutPowerSwitchingOff:=udtDeviceStatus.COIL_VALUE[9];
refIPS.xCrititicalCurrentPulseWarning:=udtDeviceStatus.COIL_VALUE[10];
refIPS.xBuzzerOn:=udtDeviceStatus.COIL_VALUE[12];
refIPS.xDisplayConnect:=udtDeviceStatus.COIL_VALUE[13];
refIPS.xADCEnable:=udtDeviceStatus.COIL_VALUE[15];
{endregion}

IF refIPS.xInterlock OR NOT refIPS.xPowerOnFeedback OR refIPS.xError OR refIPS.xOverload OR refIPS.xInputPowerOutOfLimit THEN
	refIPS.xBlocked:=TRUE;
ELSE
	refIPS.xBlocked:=FALSE;
END_IF

{region "Limit SP"}
Setting.rCurrentSP:=LIMIT(Setting.rCurrentSpMin, Setting.rCurrentSP, Setting.rCurrentSpMax);
Setting.rPowerSp:=LIMIT(Setting.rPowerSpMin, Setting.rPowerSp, Setting.rPowerSpMax);
Setting.rVoltageSP:=LIMIT(Setting.rVoltageSpMin, Setting.rVoltageSP, Setting.rPowerSpMax);
{endregion}
{region "command control"}
IF refIPS.xAutoStartCommand AND refIPS.xAutoStopCommand THEN
	refIPS.xAutoStartCommand:=FALSE;
	refIPS.xAutoStopCommand:=FALSE;		 
END_IF
IF refIPS.xManualStartCommand AND refIPS.xManualStopCommand THEN
	refIPS.xManualStartCommand:=FALSE;
	refIPS.xManualStopCommand:=FALSE;		 
END_IF
{endregion}

{region "Control"}
IF Setting.xAutoMode THEN
	IF refIPS.xAutoStartCommand THEN		 
			refIPS.xStart:=TRUE;
			refIPS.xAutoStartCommand:=FALSE;
	END_IF
	IF refIPS.xAutoStopCommand THEN
			refIPS.xStop:=TRUE;
			refIPS.xAutoStopCommand:=FALSE; 
	END_IF
ELSE
	IF refIPS.xManualStartCommand THEN 
		refIPS.xStart:=TRUE;
		refIPS.xManualStartCommand:=FALSE;
	END_IF
	IF refIPS.xManualStopCommand THEN
		refIPS.xStop:=TRUE;
		refIPS.xManualStopCommand:=FALSE;		 
	END_IF
END_IF
{endregion}

IF refIPS.xBlocked AND NOT Setting.xService THEN
	refIPS.xStart:=FALSE;
	refIPS.xStop:=TRUE;
END_IF

IF refIPS.xErrorReset  AND NOT refIPS.xTurnOn THEN
	refIPS.xErrorReset:=FALSE;
	refIPS.xError:=TRUE;
END_IF

{region "Output"}
IF refIPS.xStart THEN
	refIPS.xStart:=FALSE;
	xStart:=TRUE;		 
END_IF
IF refIPS.xStop THEN
	refIPS.xStop:=FALSE;
	xStop:=TRUE;		 
END_IF
IF refIPS.xError THEN
	refIPS.xError:=FALSE;
	xReset:=TRUE;		 
END_IF
{endregion}

END_FUNCTION_BLOCK

// Function Blocks/IPS/IPSIonModbus
FUNCTION_BLOCK IPSIonModbus
VAR_INPUT
	refModbus:	REFERENCE TO udtIPSModbus;
	Setting:	REFERENCE TO udtIPSSetting;
	rVolatgeSP:		REAL;
	rCurrentSP:		REAL;
	rPowerSP:		REAL;
END_VAR
VAR_OUTPUT
	rVoltageFeedback:	REAL;
	rCurrentFeedback:	REAL;
	rPowerFeedback:		REAL;
	sStatus:			STRING;
	xTurnOn:			BOOL;
END_VAR
VAR_IN_OUT
	xStart:BOOL;
	xStop:BOOL;
	xResetError:BOOL;
END_VAR
VAR
	Stage:				IPS_CONTROL_STAGE;
	StartStatusDelay:	TON;
	
END_VAR

{region "Input"}
refModbus.Write.strCurrentSP.sValue.INT_VALUE:=Real2Register(rValue:=rCurrentSP, iPointPosition:=Setting.CurrentPointPosition);
refModbus.Write.strVoltageSP.sValue.INT_VALUE:=Real2Register(rValue:=rVolatgeSP, iPointPosition:=Setting.VoltagePointPosition);
refModbus.Write.strPowerSP.sValue.INT_VALUE:= Real2Register(rValue:=rPowerSP, iPointPosition:=Setting.PowerPointPosition);
{endregion}
	 
{region "OPERATING LOGIC"}
CASE Stage OF
		 
	IPS_CONTROL_STAGE.WAIT:
		 IF xStart THEN
			xStart:=FALSE;
			Stage:=IPS_CONTROL_STAGE.START_PERMIT;		  
		 END_IF
		IF xStop THEN
			xStop:=FALSE;
			Stage:=IPS_CONTROL_STAGE.STOP;		 
		END_IF
			 
		IF xResetError THEN
			xResetError:=FALSE;
			Stage:=IPS_CONTROL_STAGE.ERROR_RESET;		 
		END_IF
			 
	IPS_CONTROL_STAGE.START_PERMIT:
		refModbus.Write.strCommandAndStatus.sValue.INT_VALUE:=IPS_COMMAND.START_PERMIT;
		Stage:=IPS_CONTROL_STAGE.WAIT_PERMIT_ANSWER;
			 
	IPS_CONTROL_STAGE.WAIT_PERMIT_ANSWER:
		 {info "TODO"}
		IF refModbus.Read.strCommandAndStatus.sValue.INT_VALUE = IPS_STATUS.START_PERMIT THEN
			Stage:=IPS_CONTROL_STAGE.START;
			sStatus:=TO_STRING(IPS_STATUS.START_PERMIT);
		ELSE
			Stage:=IPS_CONTROL_STAGE.ERROR;		 
		END_IF
			 
	IPS_CONTROL_STAGE.START:
		refModbus.Write.strCommandAndStatus.sValue.INT_VALUE:=IPS_COMMAND.START;
		StartStatusDelay(PT:=T#200MS,
				 			IN:=TRUE);
		IF StartStatusDelay.Q THEN
			Stage:=IPS_CONTROL_STAGE.WAIT_START_RESPONCE;
		END_IF
			 
	IPS_CONTROL_STAGE.WAIT_START_RESPONCE:
		 		StartStatusDelay(PT:=T#200MS,
				 			IN:=FALSE);
		IF refModbus.Read.strCommandAndStatus.sValue.INT_VALUE =IPS_STATUS.START_NO_ERROR THEN
			sStatus:=TO_STRING(IPS_STATUS.START_NO_ERROR);
			Stage:=IPS_CONTROL_STAGE.WAIT;
			xturnOn:=TRUE;
		ELSE
			Stage:=IPS_CONTROL_STAGE.ERROR;		 
		END_IF
			 
	IPS_CONTROL_STAGE.STOP:
		refModbus.Write.strCommandAndStatus.sValue.INT_VALUE:=IPS_COMMAND.STOP;
		Stage:=IPS_CONTROL_STAGE.WAIT_STOP_RESPONCE;
			 
	IPS_CONTROL_STAGE.WAIT_STOP_RESPONCE:
		IF refModbus.Read.strCommandAndStatus.sValue.INT_VALUE = IPS_STATUS.STOP_NO_ERROR THEN
			sStatus:=TO_STRING(IPS_STATUS.STOP_NO_ERROR);
			Stage:=IPS_CONTROL_STAGE.WAIT;
			xTurnOn:=FALSE;
		ELSE
			STAGE:=IPS_CONTROL_STAGE.ERROR;	  
		END_IF
			 
	IPS_CONTROL_STAGE.ERROR_RESET:
		refModbus.Write.strCommandAndStatus.sValue.INT_VALUE:=IPS_COMMAND.RESET_ERROR;
		Stage:=IPS_CONTROL_STAGE.WAIT_ERROR_RESET_RESPONCE;
			 
	IPS_CONTROL_STAGE.WAIT_ERROR_RESET_RESPONCE:
		 IF refModbus.Read.strCommandAndStatus.sValue.INT_VALUE = IPS_STATUS.RESET_ERROR_DONE THEN
			sStatus:=TO_STRING(IPS_STATUS.RESET_ERROR_DONE);
			Stage:=IPS_CONTROL_STAGE.WAIT;		  
		END_IF
			 
	IPS_CONTROL_STAGE.ERROR:
		 
		sStatus:=TO_STRING(refModbus.Read.strCommandAndStatus.sValue.INT_VALUE);
		xStart:=FALSE;
		xStop:=FALSE;
		Stage:=IPS_CONTROL_STAGE.WAIT;
			 
END_CASE
{endregion}

rVoltageFeedback:=GornRegister2Real(iPointPosition:=1, uiRegister:=refModbus.Read.strVoltageFeedBack.sValue.WORD_VALUE);
rCurrentFeedback:=GornRegister2Real(iPointPosition:=1, uiRegister:=refModbus.Read.strCurrenFeedback.sValue.WORD_VALUE);
rPowerFeedback:=GornRegister2Real(iPointPosition:=1, uiRegister:=refModbus.Read.strPowerFeedback.sValue.WORD_VALUE);

END_FUNCTION_BLOCK

// Function Blocks/Pumps/FVP
(*Функциональный блок для управляени форвакуумным наосос
	VERSION: 1.0
	Author: Sudalin
	DATE: 08.11.2021*)
FUNCTION_BLOCK FVP
VAR_INPUT
	refFVP: 			REFERENCE TO udtFVP;
	refFVPSetting:		REFERENCE TO udtFVPSetting;
	xPowerOnFeedback: 	BOOL; //Внешняя связь по питанию
	xTurnOn:			BOOL;//Сигнад о срабатывании контактора.
	
	xBAV1OpenedSignal:	BOOL;
	xBAV3OpenedSignal:	BOOL;
	xDoorOpenedSignal:	BOOL;
END_VAR
VAR_OUTPUT
	CommandSignal: 		BOOL;//Команда на управление 
END_VAR
VAR
END_VAR


refFVP.xPowerOnFeedBack:=xPowerOnFeedback;

refFVP.wLockStatus:=THIS^.AssebleLock();

{region "Locked status"}
IF refFVP.xInterlock OR NOT refFVP.xPowerOnFeedBack OR refFVP.wLockStatus<>0 THEN
	refFVP.xBlocked:=TRUE;
END_IF
IF refFVP.xPowerOnFeedBack AND NOT refFVP.xInterlock AND refFVP.wLockStatus = 0 THEN
	refFVP.xBlocked:=FALSE;
END_IF
{endregion}

{region "Service Mode"}
(*сервисный режим предназначен для отключения любых блокировок*)
{endregion}
{region "Lock Logic"}
IF refFVP.xBlocked AND NOT refFVPSetting.xServiceMode THEN
	refFVP.xManualCommand:=FALSE;
	refFVP.xAutoCommand:=FALSE;		 
END_IF
{endregion}
IF NOT refFVPSetting.xWithOutTurnOn THEN
	refFVP.xTurnOn:=xTurnOn;	
ELSE
	refFVP.xTurnOn:=refFVP.xStart;
END_IF


{region "Command'}
IF refFVPSetting.xAutoMode THEN
	//Автоматиечский режим
	refFVP.xManualCommand:=refFVP.xAutoCommand;
	refFVP.xStart:=refFVP.xAutoCommand;
ELSE
	//Ручной режим
	refFVP.xAutoCommand:=refFVP.xManualCommand;
	refFVP.xStart:=refFVP.xManualCommand;
END_IF
{endregion}
	 
IF NOT refFVP.xTurnOn THEN
	refFVP.wStatus:=0;
END_IF
IF refFVP.xTurnOn THEN
	refFVP.wStatus:=1;
END_IF
IF refFVP.xInterlock THEN
	refFVP.wStatus:=2;
END_IF
IF refFVP.xError THEN
	refFVP.wStatus:=3;
END_IF


CommandSignal:= refFVP.xStart;

METHOD AssebleLock : BYTE
VAR_INPUT
END_VAR
IF (THIS^.xDoorOpenedSignal OR THIS^.xBAV3OpenedSignal) AND THIS^.xBAV1OpenedSignal THEN
	AssebleLock:=1;
	RETURN;
ELSE
	AssebleLock:=0;
END_IF
END_METHOD

END_FUNCTION_BLOCK

// Function Blocks/Pumps/TMP
{attribute 'test'}
FUNCTION_BLOCK TMP
VAR_INPUT
	refTMP: 			REFERENCE TO udtTMPDigital;
	refSetting:			REFERENCE TO udtTMPDigitalSetting;
	rCameraPressure:	REAL;
	xWithSHV:			BOOL;			//Переменная конфиг
	xFVPStartSignal:	BOOL;
	xSHVOpenSignal:		BOOL;
	xNormalRelay:		BOOL;			//Реле "Нормальное состояние
	xErrorRelay:		BOOL;			//Реле "Ошибка"
	xPowerOnFeedback:	BOOL; 
END_VAR
VAR_OUTPUT
	xStart:				BOOL;
END_VAR
VAR
	StartRotateTimer:		TON;//Выход на 90hz
	StopRotatetimer:		TON;//Менее 90hz
	RotateStartSignalDelay:	TON;//Начала вращения
	RotateStopSignalDelay:	TON;//окончание вращения
	xPumpRotating:			BOOL;
	
	xStoping:			BOOL;

END_VAR


StartRotateTimer(	PT:=T#30S,
					IN:=reftmp.xStart);
StopRotatetimer(PT:=T#15S,
				IN:=NOT refTMP.xStart);

RotateStartSignalDelay(PT:=T#500MS,
						IN:=refTMP.xStart);
RotateStopSignalDelay(PT:=T#30S,
						IN:=NOT refTMP.xStart AND refTMP.xPumpRotate);
{region "Input Block"}

refTMP.xNormalOperation:=xNormalRelay;
refTMP.xPowerOnFeedBack:=xPowerOnFeedback;

{endregion}
	 	 
{region "Ack Error"}
IF xErrorRelay THEN
	refTMP.xError:= TRUE;	 
END_IF
IF refTMP.xAckError THEN
	refTMP.xAckError:=FALSE;
	refTMP.xError:=FALSE;		 
END_IF
{endregion}

refTMP.wLockResult := THIS^.AssembleLock(SHV:=xWithSHV,FVPStart:=xFVPStartSignal);
 
{region "Blocked"}
IF refTMP.xError OR refTMP.xInterlock OR NOT refTMP.xPowerOnFeedBack OR refTMP.wLockResult<>0 THEN
	refTMP.xBlocked:=TRUE;		 
END_IF
IF NOT refTMP.xError AND NOT refTMP.xInterlock AND refTMP.xPowerOnFeedBack AND refTMP.wLockResult=0 THEN
	refTMP.xBlocked:=FALSE;		 
END_IF
{endregion}

{region "Blocked Logic"}
IF refTMP.xBlocked AND NOT refSetting.xServiceMode THEN
	refTMP.xManualCommand:=FALSE;
	refTMP.xAutoCommand:=FALSE;	 
END_IF
{endregion}
	 
{region "Auto/Man Command"}
IF refSetting.xAutoMode THEN
//Автоматический режим
	refTMP.xManualCommand:=refTMP.xAutoCommand;
	refTMP.xStart:=refTMP.xAutoCommand;
ELSE
//Ручной режим 
	refTMP.xAutoCommand:=refTMP.xManualCommand;
	refTMP.xStart:=refTMP.xManualCommand;
END_IF
{endregion}
{region "Status"}
	refTMP.xMore90hzRotate:=StatustimerLogic(StartQ:=StartRotateTimer.Q, StopQ:=StopRotateTimer.Q);
	refTMP.xPumpRotate:=RotateSignalAssemble(DelayStartQ:=RotateStartSignalDelay.Q, FullStopQ:=RotateStopSignalDelay.Q);
{endregion}
	 
StatusAssemble(	refErrJustOccured:= refTMP.errJustOccured,
				refErrPumpIsDecelerating:= refTMP.errPumpIsDecelerating,
				refErrPumpStandstill:=refTMP.errPumpStandstill,
				xError:=refTMP.xError,
				refJustAfterStart:=refTMP.xJustAfterStart,
				refJustAfterStop:=refTMP.xJustAfterStop,
				xMore90hzRotate:=refTMP.xMore90hzRotate,
				xNormalOperation:=refTMP.xNormalOperation,
				refPumpIsAccelerating:=refTMP.xPumpIsAccelerating,
				refPumpIsDecelerating:=refTMP.xPumpIsDecelerating,
				refPumpNormalOperatingMode:=refTMP.xPumpNormalOperatingMode,
				refPumpNotOperating:=refTMP.xPumpNotOperating,
				xPumpRotate:=refTMP.xPumpRotate,
				xStart:=refTMP.xStart 
				
	);
IF refTMP.xPumpNotOperating AND NOT refTmp.xPumpIsDecelerating THEN
	refTMP.wStatus :=0;
END_IF
IF refTMP.xPumpNormalOperatingMode THEN
	refTMP.wStatus:=1;
END_IF
IF refTMP.xInterlock THEN
	refTMP.wStatus:=2;
END_IF
IF refTMP.xError THEN
	refTMP.wStatus:=3;
END_IF
IF refTmp.xPumpIsDecelerating THEN
	refTMP.wStatus:=4;
END_IF
IF refTMP.xPumpIsAccelerating THEN
	refTMP.wStatus:=5;
END_IF

xStart:=refTMP.xStart;

METHOD AssembleLock : BYTE
VAR_INPUT
	SHV: BOOL;
	FVPStart: BOOL;
END_VAR
IF SHV THEN
	AssembleLock:=THIS^.AssembleLockWithSHV(FVPStart);
ELSE
	AssembleLock:=0;
END_IF
END_METHOD

METHOD PRIVATE AssembleLockWithSHV : BYTE
VAR_INPUT
	FVPStart: BOOL;
END_VAR
IF NOT FVPStart THEN
	AssembleLockWithSHV:=1;
	RETURN;
ELSIF THIS^.xSHVOpenSignal AND THIS^.rCameraPressure>refSetting.rMinimalCameraPressure THEN
	AssembleLockWithSHV:=2;
	RETURN;
ELSE
	AssembleLockWithSHV:=0;
END_IF
END_METHOD

METHOD RotateSignalAssemble : BOOL
VAR_INPUT
	DelayStartQ:			BOOL;//Сигнал о задержке после старта
	FullStopQ:				BOOL;//Сигнал о срабатывании таймера после стопа
END_VAR
IF DelayStartQ THEN
	RotateSignalAssemble:=TRUE;
END_IF
IF FullStopQ THEN
	RotateSignalAssemble:=FALSE;
END_IF
END_METHOD

METHOD StatusAssemble : BOOL
VAR_INPUT
	refPumpNotOperating:		 	REFERENCE TO BOOL;	
	refPumpIsDecelerating: 		REFERENCE TO BOOL;
	refJustAfterStop:				REFERENCE TO BOOL;
	refJustAfterStart:			REFERENCE TO BOOL;
	refPumpIsAccelerating:		REFERENCE TO BOOL;
	refPumpNormalOperatingMode: 	REFERENCE TO BOOL;
	refErrPumpStandstill:			REFERENCE TO BOOL;
	refErrPumpIsDecelerating:		REFERENCE TO BOOL;
	refErrJustOccured:				REFERENCE TO BOOL;
	
	xStart:				BOOL;//сигнал на старт.стоп
	xPumpRotate:		BOOL;
	xMore90hzRotate:	BOOL;
	xError:				BOOL;
	xNormalOperation:	BOOL;
END_VAR
IF NOT xStart AND NOT xPumpRotate AND NOT xMore90hzRotate AND NOT xError AND NOT xNormalOperation THEN
 	refPumpNotOperating:=TRUE;
ELSE
	refPumpNotOperating:=FALSE;
END_IF

IF NOT xStart AND xPumpRotate AND NOT xMore90hzRotate AND NOT xNormalOperation AND NOT xError THEN
	refPumpIsDecelerating:=TRUE;
ELSE	
	refPumpIsDecelerating:=FALSE;
END_IF

IF NOT xStart AND xPumpRotate AND xMore90hzRotate AND NOT xNormalOperation AND NOT xError THEN
	refJustAfterStop:=TRUE;
ELSE
	refJustAfterStop:=FALSE;
END_IF

IF xStart AND NOT xPumpRotate AND NOT xMore90hzRotate AND NOT xNormalOperation AND NOT xError THEN
		refJustAfterStart:=TRUE;
ELSE
		refJustAfterStart:=FALSE;		
END_IF


IF xStart AND xPumpRotate AND NOT xMore90hzRotate AND NOT xNormalOperation AND NOT xError THEN
	refPumpIsAccelerating:=TRUE;
ELSE
	refPumpIsAccelerating:=FALSE;	
END_IF

IF xStart AND xPumpRotate AND xMore90hzRotate AND xNormalOperation AND NOT xError THEN
	refPumpNormalOperatingMode:=TRUE;
ELSE
	refPumpNormalOperatingMode:=FALSE;
END_IF

IF  NOT xPumpRotate AND xMore90hzRotate AND NOT xNormalOperation AND xError THEN
	refErrPumpStandstill:=TRUE;
ELSE
	refErrPumpStandstill:=FALSE;
END_IF

IF  xPumpRotate AND NOT xMore90hzRotate AND NOT xNormalOperation AND xError THEN
	refErrPumpIsDecelerating:=TRUE;
ELSE
	refErrPumpIsDecelerating:=FALSE;
END_IF

IF   xPumpRotate AND xMore90hzRotate AND NOT xNormalOperation AND xError THEN
	refErrJustOccured:=TRUE;
ELSE
	refErrJustOccured:=FALSE;
END_IF
END_METHOD

METHOD StatusTimerLogic : BOOL;
VAR_INPUT
	StartQ:BOOL;
	StopQ:BOOL;
END_VAR
IF StartQ THEN
	StatusTimerLogic:=TRUE;
END_IF
IF StopQ THEN
	StatusTimerLogic:=FALSE;
END_IF
END_METHOD

END_FUNCTION_BLOCK

// Function Blocks/Pumps/TMPPfifer
FUNCTION_BLOCK TMPPfifer
VAR_INPUT
	refTMP: 			REFERENCE TO udtTMPDigital;
	refSetting:			REFERENCE TO udtTMPDigitalSetting;
	
	xWithSHV:			BOOL;			//Переменная конфиг
    xPowerOnFeedback:	BOOL;
END_VAR
VAR_OUTPUT
	xStart: BOOL;
END_VAR
VAR
	StartTimer:TON;
	StopTimer: TON;
	WasStart:	BOOL;
END_VAR

StartTimer(IN:=refTMP.xStart,
			PT:=T#8M);
{region "Input Block"}
StopTimer(IN:=NOT refTMP.xStart AND WasStart,
			PT:=T#2M);

refTMP.xPowerOnFeedBack:=xPowerOnFeedback;

{endregion}
	 	 



 
{region "Blocked"}
IF refTMP.xError OR refTMP.xInterlock OR NOT refTMP.xPowerOnFeedBack OR refTMP.wLockResult<>0 THEN
	refTMP.xBlocked:=TRUE;		 
END_IF
IF NOT refTMP.xError AND NOT refTMP.xInterlock AND refTMP.xPowerOnFeedBack AND refTMP.wLockResult=0 THEN
	refTMP.xBlocked:=FALSE;		 
END_IF
{endregion}

{region "Blocked Logic"}
IF refTMP.xBlocked AND NOT refSetting.xServiceMode THEN
	refTMP.xManualCommand:=FALSE;
	refTMP.xAutoCommand:=FALSE;	 
END_IF
{endregion}
	 
{region "Auto/Man Command"}
IF refSetting.xAutoMode THEN
//Автоматический режим
	refTMP.xManualCommand:=refTMP.xAutoCommand;
	refTMP.xStart:=refTMP.xAutoCommand;
ELSE
//Ручной режим 
	refTMP.xAutoCommand:=refTMP.xManualCommand;
	refTMP.xStart:=refTMP.xManualCommand;
END_IF
{endregion}

IF StartTimer.Q THEN
	WasStart:=TRUE;
END_IF
IF StopTimer.Q THEN
	WasStart:=FALSE;
END_IF
refTMP.xPumpIsAccelerating:= refTMP.xStart AND NOT StartTimer.Q;
refTMP.xPumpNormalOperatingMode:=refTMP.xStart AND StartTimer.Q;
refTMP.xNormalOperation:=refTMP.xPumpNormalOperatingMode;
refTMP.xPumpIsDecelerating:=NOT refTMP.xStart AND NOT StopTimer.Q AND WasStart;
refTMP.xPumpNotOperating:=(NOT refTMP.xStart AND StopTimer.Q) OR NOT WasStart;

IF refTMP.xPumpNotOperating  THEN
	refTMP.wStatus :=0;
END_IF
IF refTMP.xPumpNormalOperatingMode THEN
	refTMP.wStatus:=1;
END_IF
IF refTMP.xInterlock THEN
	refTMP.wStatus:=2;
END_IF
IF refTMP.xError THEN
	refTMP.wStatus:=3;
END_IF
IF refTmp.xPumpIsDecelerating THEN
	refTMP.wStatus:=4;
END_IF
IF refTMP.xPumpIsAccelerating THEN
	refTMP.wStatus:=5;
END_IF

xStart:=refTMP.xStart;

END_FUNCTION_BLOCK

// Function Blocks/RRG/fbRRG
FUNCTION_BLOCK fbRRG
VAR_INPUT
	RRG: REFERENCE TO udtRRG;
	Setting: REFERENCE TO udtRRGSetting;
	Interlock: BOOL;
END_VAR
VAR_OUTPUT
	xError: BOOL;
END_VAR
VAR
	oldSP: REAL:=0.0;
END_VAR

IF NOT Setting.xAutoMode THEN
	RRG.rManualValueSP:= LIMIT(Setting.rMinValue, RRG.rManualValueSP, Setting.rMaxValue);
	RRG.rAutoValueSP:= RRG.rManualValueSP;
	RRG.rValueSP:=RRG.rManualValueSP;
END_IF

IF Setting.xAutoMode THEN
	RRG.rAutoValueSP := LIMIT(Setting.rMinValue, RRG.rAutoValueSP, Setting.rMaxValue);
	RRG.rManualValueSP:=RRG.rAutoValueSP;
	RRG.rValueSP:=RRG.rAutoValueSP;
END_IF

IF NOT Setting.xService AND Interlock THEN
	RRG.rValueSP:=0.0;
END_IF

IF oldSP <>RRG.rValueSP THEN
	RRG.trigNewSp:=TRUE;
	oldSP:=RRG.rValueSP;
ELSE
	RRG.trigNewSp:=FALSE;
END_IF




RRG.xError:=RRG.xLowGasFlow;
xError:=RRG.xError;

END_FUNCTION_BLOCK

// Function Blocks/RRG/fbRRGModbus
FUNCTION_BLOCK fbRRGModbus
VAR_INPUT
	Setting: 	REFERENCE TO udtRRGSetting;
	Modbus: 	REFERENCE TO udtRRGModbus;
	RRG: 		REFERENCE TO udtRRG;
END_VAR
VAR_OUTPUT
END_VAR
VAR
END_VAR

Modbus.GasFlowSPWrite:=ConvertValueSPtoModbusData();
RRG.rValueFeedback:=ConvertModbusValueFbTovalueFb();
AssembleStatusFromFieldStatus2();
UnmarshalModbusFlagStatus1ToRRGFeedback();

METHOD AssembleStatusFromFieldStatus2
VAR_INPUT
END_VAR
RRG.xLowGasFlow:=Modbus.FlagState2.Flags.LowGasFlow;
RRG.xValveMode:=Modbus.FlagState2.Flags.ValveMode;
RRG.xRegMode:=Modbus.FlagState2.Flags.RegMode;
RRG.xOnlyRDG:=Modbus.FlagState2.Flags.RDGOnly;
RRG.xOnlyRRG:=Modbus.FlagState2.Flags.RRGOnly;

RRG.xValveCloseState:= Modbus.FlagState2.Flags.StateBit5 AND NOT Modbus.FlagState2.Flags.StateBit6;
RRG.xValveOpenState:= NOT Modbus.FlagState2.Flags.StateBit5 AND  Modbus.FlagState2.Flags.StateBit6;
RRG.xValveRegModeState:= NOT Modbus.FlagState2.Flags.StateBit5 AND NOT Modbus.FlagState2.Flags.StateBit6;
END_METHOD

METHOD ConvertModbusSPFeedbackToSPfeedback : REAL
VAR_INPUT
END_VAR
ConvertModbusSPFeedbackToSPfeedback:=(Setting.rMaxValue-Setting.rMinValue)*(Modbus.GasFlowSPRead/100);
END_METHOD

METHOD ConvertModbusValueFbTovalueFb : Real
VAR_INPUT
END_VAR
ConvertModbusValueFbTovalueFb:=((DWORD_TO_REAL(WORD_TO_DWORD(Modbus.GasFlowFB)))/(100*100))*(Setting.rMaxValue-Setting.rMinValue);
END_METHOD

METHOD ConvertValueSPtoModbusData : WORD
VAR_INPUT
END_VAR
ConvertValueSPtoModbusData:=REAL_TO_WORD((RRG.rValueSP/(Setting.rMaxValue-Setting.rMinValue))*100*100);
END_METHOD

METHOD UnmarshalModbusFlagStatus1ToRRGFeedback
VAR_INPUT
END_VAR
RRG.xDigitalInputFeedback := Modbus.FlagState1_Read.Flags.DigitalInput;
RRG.xRepaireModeFeedback:= Modbus.FlagState1_Read.Flags.RepareBit;
RRG.xRRGModeFeedback:=Modbus.FlagState1_Read.Flags.RRGMode;

RRG.xValveOpenFeedback:=Modbus.FlagState1_Read.Flags.StateBit2 AND NOT Modbus.FlagState1_Read.Flags.StateBit3;
RRG.xValveCloseFeedback:=NOT Modbus.FlagState1_Read.Flags.StateBit2 AND  Modbus.FlagState1_Read.Flags.StateBit3;
RRG.xValveRegModeFeedback:=NOT Modbus.FlagState1_Read.Flags.StateBit2 AND NOT Modbus.FlagState1_Read.Flags.StateBit3;
END_METHOD

END_FUNCTION_BLOCK

// Function Blocks/Shutter/fbShutter
FUNCTION_BLOCK fbShutter
VAR_INPUT
	Shutter: 		REFERENCE TO udtShutter;
	Setting:		REFERENCE TO udtShutterSetting;
	ShutterOpened:	BOOL;
	Interlock:		BOOL;
END_VAR
VAR_OUTPUT
	OpenSignal: 	BOOL;
	CloseSignal:	BOOL;
END_VAR
VAR
END_VAR


Shutter.Interlock:=Interlock;


IF Setting.AutoMode THEN
	Shutter.ManualCommand:=Shutter.AutoCommand;
	Shutter.FinallyCommand:=Shutter.AutoCommand;
END_IF

IF (NOT Setting.AutoMode) THEN
	Shutter.AutoCommand:=Shutter.ManualCommand;
	Shutter.FinallyCommand:=Shutter.ManualCommand;
END_IF

(*
	При FinallyCommand = true заслонка открывает
	При FinallyCommand = false заслонка закрыватся
*)


Shutter.AutoMode:=Setting.AutoMode;
IF Shutter.FinallyCommand AND NOT Shutter.ShutterOpened THEN
	Shutter.OpenCommand:=TRUE;

ELSIF Shutter.FinallyCommand AND  Shutter.ShutterOpened THEN
	Shutter.OpenCommand:=FALSE;
END_IF


IF NOT Shutter.FinallyCommand AND Shutter.ShutterOpened THEN
	Shutter.CloseCommand:=TRUE;
	
ELSIF NOT Shutter.FinallyCommand AND NOT Shutter.ShutterOpened THEN
	Shutter.CloseCommand:=FALSE;
END_IF

IF Setting.WithoutEnder AND Shutter.FinallyCommand THEN
	Shutter.ShutterOpened:=TRUE;
ELSIF Setting.WithoutEnder AND NOT Shutter.FinallyCommand THEN
	Shutter.ShutterOpened:=FALSE;
ELSE
	Shutter.ShutterOpened:=ShutterOpened;
END_IF

IF Setting.RemoteMode THEN
	OpenSignal:=Shutter.OpenCommand;
	CloseSignal:=Shutter.CloseCommand;
ELSE
	Shutter.OpenCommand:=FALSE;
	Shutter.CloseCommand:=FALSE;
	Shutter.ManualCommand:=FALSE;
	SHutter.AutoCommand:=FALSE;
	OpenSignal:=FALSE;
	CloseSignal:=FALSE;	
END_IF

END_FUNCTION_BLOCK

// Function Blocks/TRM_View/MC_Heater
FUNCTION_BLOCK MC_Heater
VAR_INPUT
	refHeater:				REFERENCE TO udtTRMHeaterView; 			//сонвоной блок визуализации и контроля
	refInput_1:				REFERENCE TO udtTRMInputView;			//Данные первого канала
	refInput_2:				REFERENCE TO udtTRMInputView;			//Данные второго канала
	refRegulator_1:			REFERENCE TO udtTRMRegulatorView;		//Данные первого регулятора
	refRegulator_2:			REFERENCE TO udtTRMRegulatorView;		//Данные второго регулятора
	refOutput_1:			REFERENCE TO udtTRMOutput;				//Данные первого выхода
	refOutput_2:			REFERENCE TO udtTRMOutput;				//Данные второго выхода
	refChannel_1:			REFERENCE TO udtTRMChannelView;			//Данные первого канала
	refChannel_2:			REFERENCE TO udtTRMChannelView;			//Данные второго канала
	refOperating:			REFERENCE TO udtTRMOperatingView;		//Оперативные данные
	refTechnologOperation:	REFERENCE TO udtTRMTechnologOperation;	//Составление программы оператора
	
	xInputSaveEvent: 		REFERENCE TO BOOL;
	xRegulatorSaveEvent:	REFERENCE TO BOOL;
	xOutputSaveEvent:		REFERENCE TO BOOL;
	xProgramStepSaveEvent:	REFERENCE TO BOOL;
	xStartStopEvent:		REFERENCE TO BOOL;
	xSaveOperationProgram:	REFERENCE TO BOOL;
	
	xPower:			BOOL;
	xInterlock:		BOOL;
END_VAR
VAR_OUTPUT
	xBlocked: BOOL;
	
END_VAR
VAR
	Channel:				MC_TRMChannel;
	Input:					MC_TRMInput;
	Regulator:  			MC_TRMRegulator;
	Output:					MC_TRMOutput;
	Operating:				MC_TRMOperating;
	ProgramOfTechnolog:		MC_TRMProgramOfTechnolog;
	
	xInit:			BOOL:=FALSE;//Флаг инициализации
END_VAR

IF NOT xInit THEN

	xInit:=TRUE;
	(*Инициализация сохранения*)
	
	Regulator.xSaveSignal 	REF= refHeater.xSaveRegulator;
	
	xSaveOperationProgram 	REF= refTechnologOperation.xSaveEvent;
	
END_IF
{region "INPUT"}
refHeater.xPowerOn:=xPower;
refHeater.xInterlock:=xInterlock;

{endregion}
	Input(refInput:=refInput_1);
	Input(refInput:=refInput_2);
	Regulator(refRegulator:=refRegulator_1);
	Regulator(refRegulator:=refRegulator_1);
	Output(refOutput:=refOutput_1);
	Output(refOutput:=refOutput_2);
	Operating(refOperating:=refOperating);
	ProgramOfTechnolog(refTechnolog:=refTechnologOperation);

(*{region "Programm Limit"}
refHeater.ProgrammNoSP:=LIMIT(0, refHeater.ProgrammNoSP, 11);
refHeater.ProgramStepNoFb:=LIMIT(0, refHeater.ProgramStepNoSP, 9);
{endregion}*)
	 
{region "BLOCKED STATUS"}
IF refHeater.xInterlock OR NOT refHeater.xPowerOn THEN
	refHeater.xBlocked:=TRUE;		 
END_IF
{endregion}
	 
{region "Channel logic}
Channel(udtChannel:=refChannel_1);
Channel(udtChannel:=refChannel_2);
{endregion}

(*Сохранение шага и программы старта если регулятор выключен*)
IF refHeater.xSaveStartProgramAndStep AND (refHeater.Status = TRMObjectState.Stop OR refHeater.Status = TRMObjectState.StopAfterComplite) THEN
	refHeater.xSaveStartProgramAndStep:=FALSE;
	xProgramStepSaveEvent:=TRUE;
ELSE
	refHeater.xSaveStartProgramAndStep:=FALSE;
END_IF

	 
IF refHeater.xAutoMode THEN
	IF refHeater.xAutoStart THEN
		refHeater.xAutoStart:=FALSE;
		refOperating.StartProcessSignal:=TRMStartSignal.RUN;
		xStartStopEvent:=TRUE;
	END_IF
	IF refHeater.xAutoStop THEN
		refheater.xAutoStop:=FALSE;
		refOperating.StartProcessSignal:=TRMStartSignal.STOP;
		xStartStopEvent:=TRUE;
	END_IF
ELSE
	IF refHeater.xManualStart THEN
		refHeater.xManualStart:=FALSE;
		refOperating.StartProcessSignal:=TRMStartSignal.RUN;
		xStartStopEvent:=TRUE;
	END_IF
	IF refHeater.xManualStop THEN
		refHeater.xManualStop:=FALSE;
		refOperating.StartProcessSignal:=TRMStartSignal.STOP;
		xStartStopEvent:=TRUE;
	END_IF
END_IF

{region "OUTPUT"}
xBlocked:=refHeater.xBlocked;
{endregion}

END_FUNCTION_BLOCK

// Function Blocks/TRM_View/MC_TRMChannel
FUNCTION_BLOCK MC_TRMChannel
VAR_INPUT
	udtChannel:				REFERENCE TO udtTRMChannelView;
	xProgramMode:			BOOL; // Разрешение на уставку 0 - ручной режим ; 1-программа
	xBlocked:				BOOL; // Статус блокировки
END_VAR
VAR_OUTPUT
	
END_VAR
VAR
END_VAR

//TODO: SaveSignal

END_FUNCTION_BLOCK

// Function Blocks/TRM_View/MC_TRMInput
FUNCTION_BLOCK MC_TRMInput
VAR_INPUT
	refInput:	REFERENCE TO udtTRMInputView;
	
END_VAR
VAR_OUTPUT
END_VAR
VAR
END_VAR

{region "Limit SP"}
refInput.CorrectionOfCharacteresticShift:=LIMIT(refInput.CorrectionOfCharacteristicShiftMin, refInput.CorrectionOfCharacteresticShift, refInput.CorrectionOfCharacteristicShiftMax);
refInput.CorrectionOfInclineCharacteristic:=LIMIT(refInput.CorrectionOfInclineCharacteristicMin, refInput.CorrectionOfInclineCharacteristic, refInput.CorrectionOfInclineCharacterisitcMax);
refInput.DigitalFilterLine:=LIMIT(refInput.DigitalFilterLineMin, refInput.DigitalFilterLine, refInput.DigitalFilterLineMax);
refInput.DigitalFiltertimeConst:=LIMIT(refInput.DigitalFilterConstMin, refInput.DigitalFiltertimeConst, refInput.DigitalFilterConstMax);
refInput.HightEdgeSensoreChange:=LIMIT(refInput.HightEdgeSensoreChangeMin, refInput.HightEdgeSensoreChange, refInput.HightEdgeSensoreChangeMax);
refInput.LowEdgeSensoreChange:=LIMIT(refInput.LowEdgeSensoreChangeMin, refInput.LowEdgeSensoreChange, refInput.LowEdgeSensoreChangeMax);
{endregion}

END_FUNCTION_BLOCK

// Function Blocks/TRM_View/MC_TRMRegulator
FUNCTION_BLOCK MC_TRMRegulator
VAR_INPUT
	refRegulator: 	REFERENCE TO udtTRMRegulatorView;
	xSaveSignal:	REFERENCE TO BOOL;	
END_VAR
VAR_OUTPUT
END_VAR
VAR
END_VAR

{region "LIMIT"}
	refRegulator.PIDRegualtor.MinIntegralLimit:=LIMIT(refRegulator.PIDRegualtor.MinIntegralLimitMin, refRegulator.PIDRegualtor.MinIntegralLimit, refRegulator.PIDRegualtor.MinIntegralLimitMax);
	refRegulator.PIDRegualtor.MaxIntegralLimit:=LIMIT(refRegulator.PIDRegualtor.MaxIntegralLimitMax, refRegulator.PIDRegualtor.MaxIntegralLimit, refRegulator.PIDRegualtor.MaxIntegralLimitMax);
{endregion}
	 
{region "Save signal"}
IF xSaveSignal THEN
	xSaveSignal:=FALSE;
	refRegulator.xSaveEvent:=TRUE;		 
END_IF
{endregion}

END_FUNCTION_BLOCK

// Function Blocks/TRM_View/MC_TRMOutput
FUNCTION_BLOCK MC_TRMOutput
VAR_INPUT
	refOutput:		REFERENCE TO udtTRMOutput;

	
END_VAR
VAR_OUTPUT
END_VAR
VAR
END_VAR

{region "LIMIT"}
refOutput.MaxOutputPower:=LIMIT(refOutput.MaxOutputPowerMin, refOutput.MaxOutputPower, refOutput.MaxOutputPowerMax);
refOutput.MaxSpeedOutputPowerSpeed:=LIMIT(refOutput.MaxSpeedOutputPowerSpeedMin, refOutput.MaxSpeedOutputPowerSpeed, refOutput.MaxSpeedOutputPowerSpeedMax);
refOutput.MinOutputPower:=LIMIT(refOutput.MinOutputPowerMin, refOutput.MinOutputPower, refOutput.MinOutputPowerMax);
{endregion}

END_FUNCTION_BLOCK

// Function Blocks/TRM_View/MC_TRMOperating
FUNCTION_BLOCK MC_TRMOperating
VAR_INPUT
	refOperating:			REFERENCE TO udtTRMOperatingView;
	
END_VAR
VAR_OUTPUT
END_VAR
VAR
END_VAR

refOperating.ProgrammNoSP:=LIMIT(1, refOperating.ProgrammNoSP, 12);
refOperating.ProgramStepNoSP:=LIMIT(1, refOperating.ProgramStepNoSP,10);

END_FUNCTION_BLOCK

// Function Blocks/TRM_View/MC_TRMProgramOfTechnolog
FUNCTION_BLOCK MC_TRMProgramOfTechnolog
VAR_INPUT
	refTechnolog:				REFERENCE TO udtTRMTechnologOperation;
END_VAR
VAR_OUTPUT
END_VAR
VAR
END_VAR

refTechnolog.ProgramNo:=LIMIT(1, refTechnolog.ProgramNo, 12);
refTechnolog.StepNo:=LIMIT(1, refTechnolog.StepNo,10);


IF refTechnolog.xLoadProgram THEN
	refTechnolog.xLoadProgram := FALSE;
	refTechnolog.ViewTechnologOperationProgram:=refTechnolog.TechnologOperationProgram[refTechnolog.ProgramNo-1];

END_IF

IF refTechnolog.xSaveProgram THEN
	refTechnolog.xSaveProgram:=FALSE;
	refTechnolog.xSaveEvent:=TRUE;
	refTechnolog.TechnologOperationProgram[refTechnolog-1]:=refTechnolog.ViewTechnologOperationProgram;
END_IF

refTechnolog.ViewTechnologOperationProgramStep REF= refTechnolog.ViewTechnologOperationProgram.Step[refTechnolog.StepNo-1];
refTechnolog.ViewStepSetpoint REF= refTechnolog.ViewTechnologOperationProgram.StepSetPoint[refTechnolog.StepNo-1];

END_FUNCTION_BLOCK

// Function Blocks/VacuumSensore/VacuumSensore
FUNCTION_BLOCK VacuumSensore
VAR_INPUT
	rVoltage: REAL;
	refVacuumSensore: REFERENCE TO udtPressureSensore;
	refvacuumSensoreSetting: REFERENCE TO udtPressureSensoreSettiing;
END_VAR
VAR_OUTPUT
	xError:	BOOL;
	Pressure: REAL;
END_VAR
VAR

END_VAR

{region "INPUT SIGNAL"}
IF rVoltage > refvacuumSensoreSetting.rVolageDeathband THEN
	refVacuumSensore.rVolatgeSignal:=rVoltage;
	refVacuumSensore.xError:=FALSE;
ELSIF rVoltage<refvacuumSensoreSetting.rVolageDeathband AND rVoltage > 1.3 THEN
	refVacuumSensore.rVolatgeSignal:=refvacuumSensoreSetting.rVolageDeathband;
	refVacuumSensore.xError:=FALSE;
ELSE
	refVacuumSensore.rVolatgeSignal:=refvacuumSensoreSetting.rVolageDeathband;
	refVacuumSensore.xError:=TRUE;
END_IF
{endregion}
	 
{region "VacuumCalc"}
CASE refvacuumSensoreSetting.enumPressureUnit OF
		 PRESSURE_UNIT.mBar:
			  refVacuumSensore.rPressure:=THIS^.CalcPressure(rVoltage:= refVacuumSensore.rVolatgeSignal,
					   			rKVoltage:= refvacuumSensoreSetting.rKVoltage,
								rKPressure:=refvacuumSensoreSetting.rKMBar);
			refVacuumSensore.sUnit:='mBar';
		PRESSURE_UNIT.Pascal:
			  refVacuumSensore.rPressure:=THIS^.CalcPressure(rVoltage:= refVacuumSensore.rVolatgeSignal,
					   			rKVoltage:= refvacuumSensoreSetting.rKVoltage,
								rKPressure:=refvacuumSensoreSetting.rKPa);
			refVacuumSensore.sUnit:='Pa';
		PRESSURE_UNIT.Torr:
			  refVacuumSensore.rPressure:=THIS^.CalcPressure(rVoltage:= refVacuumSensore.rVolatgeSignal,
					   			rKVoltage:= refvacuumSensoreSetting.rKVoltage,
								rKPressure:=refvacuumSensoreSetting.rKTorr);
			refVacuumSensore.sUnit:='Torr';
		ELSE
			refvacuumSensoreSetting.enumPressureUnit:= PRESSURE_UNIT.mBar;
			 
END_CASE
{endregion}
{region "Simpulation"}
IF refvacuumSensoreSetting.xSimMode THEN
	refVacuumSensore.rPressure:=refvacuumSensoreSetting.rSimValue;		 
END_IF
{endregion}
Pressure:= refVacuumSensore.rPressure;

METHOD PRIVATE CalcPressure : REAL
VAR_INPUT
	rVoltage:	REAL; // Значение напряжения
	rKVoltage:	REAL; // Коэффициент напряжения
	rKPressure: REAL; // Вчитаемое
END_VAR
VAR_STAT
	tempExponent: REAL; // Переменная дл расчтеа экспоненты
END_VAR
tempExponent:=((rKVoltage*rVoltage)-rKPressure);
CalcPressure:= EXPT(10.0, tempExponent);
END_METHOD

END_FUNCTION_BLOCK

// Function Blocks/Valves/Valve
FUNCTION_BLOCK Valve
VAR_INPUT
	xOpened: 			BOOL;
	xClosed:			BOOL;
	refValve:			REFERENCE TO udtValve;	
	refValveSetting:	REFERENCE TO udtValveSetting;
END_VAR
VAR_OUTPUT
	xOpen:		BOOL;
	xClose:		BOOL;
	xError:		BOOL;
	
END_VAR
VAR
	OpenCloseTimer: TON;
	xInit:	BOOL;
	xStartTimerSignal: BOOl;
END_VAR


	OpenCloseTimer.PT:=refValveSetting.tGripTime;


OpenCloseTimer(IN:=xStartTimerSignal);


IF refValveSetting.xOnlycCloseEnderMode THEN
	refvalve.xClosed:=xClosed;
	refValve.xOpened:=NOT refValve.xClosed;
ELSIF refValveSetting.xWithoutEnderMode THEN
	refValve.xClosed:= NOT refValve.xOpen;
	refValve.xOpened:=refValve.xOpen;
ELSE
	refValve.xOpened:=xOpened;
	refvalve.xClosed:=xClosed;
END_IF





IF (refValve.xInterlock AND NOT refValveSetting.xServiceMode) OR refValve.xError THEN
	refValve.xManualCommand:=FALSE;
	refValve.xAutoCommand:=FALSE;
	refValve.xBlocked:=TRUE;
ELSE
	refValve.xBlocked:=FALSE;
END_IF


IF refValveSetting.xAutoMode THEN
	refValve.xManualCommand:=refValve.xAutoCommand;
	refValve.xOpen:=refValve.xAutoCommand;
	refValve.xClose:= NOT refValve.xAutoCommand;
END_IF

IF NOT refValveSetting.xAutoMode THEN
	refValve.xAutoCommand:=refvalve.xManualCommand;
	refvalve.xOpen:=refValve.xManualCommand;
	refValve.xClose:=NOT refValve.xManualCommand;
END_IF

IF (NOT refValve.xOpened AND NOT refValve.xClosed) OR (refvalve.xOpen AND NOT refvalve.xOpened) OR (refvalve.xClose AND NOT refValve.xClosed) THEN
	xStartTimerSignal:=TRUE;
ELSE
	xStartTimerSignal:=FALSE;
END_IF 


IF OpenCloseTimer.Q THEN
	refValve.xError:=TRUE;
ELSE
	refValve.xError:=FALSE;
END_IF

IF refValve.xClosed THEN
	refValve.wVavleStatus:=0;
END_IF
IF refValve.xOpened THEN
	refValve.wVavleStatus:=1;
END_IF
IF refValve.xInterlock THEN
	refValve.wVavleStatus:=2;
END_IF
IF refValve.xError THEN
	refValve.wVavleStatus:=3;
END_IF


xOpen:=refValve.xOpen;
xClose:=refValve.xClose;
xError:=refValve.xError;

END_FUNCTION_BLOCK

// Function Blocks/Valves/ValvesInterlock
FUNCTION_BLOCK ValvesInterlock
VAR_INPUT
	BAV1: REFERENCE TO udtValve;
	BAV2: REFERENCE TO udtValve;
	BAV3: REFERENCE TO udtvalve;
	SHV:  REFERENCE TO udtValve;
	CameraPressure:	REAL;
	SHVAccessPresure:	REAL; //Давление в камере ниже которого можно открывать SHV
	TMPRunSignal:	BOOL;
	LowPressureRelaySignal: BOOL;
END_VAR
VAR_OUTPUT
END_VAR
VAR
	BAV1LowPressureInterlock: BOOL;
	BAV2LowPressureInterlock: BOOL;
	BAV3LowPressureInterlock: BOOL;
	BAV1LockedBAV3Opened: BOOL;
	BAV2LockedBAV3opened: BOOL;
	BAV3LockedBAV1Opened: BOOL;
	BAV3LockedBAV2Opened: BOOL;
	BAV3LockedSHVOpened:	BOOL;
END_VAR

BAV1LowPressureInterlock:=	LowPressureInterlock();
BAV2LowPressureInterlock:=	LowPressureInterlock();
BAV3LowPressureInterlock:=	LowPressureInterlock();

BAV1LockedBAV3Opened:=AnotherValveOpenInterlock(OpenSignalValveLocker:=BAV3.xOpened);
BAV2LockedBAV3Opened:=AnotherValveOpenInterlock(OpenSignalValveLocker:=BAV3.xOpened);

BAV3LockedBAV1Opened:=AnotherValveOpenInterlock(OpenSignalValveLocker:=BAV1.xOpened);
BAV3LockedBAV2Opened:=AnotherValveOpenInterlock(OpenSignalValveLocker:=BAV2.xOpened);
BAV3LockedSHVOpened:=AnotherValveOpenInterlock(OpenSignalValveLocker:=SHV.xOpened);

BAV1.wInterlockStatus:=AssembleValveStatus(	LowPressureInterlock:=BAV1LowPressureInterlock,
											AnotherValveOpenInterlock:=BAV1LockedBAV3Opened,
											Interlock:=BAV1.xInterlock);
											
BAV2.wInterlockStatus:=AssembleValveStatus (LowPressureInterlock:=BAV2LowPressureInterlock,
											AnotherValveOpenInterlock:=BAV2LockedBAV3opened,
											Interlock:=BAV2.xInterlock);

BAV3.wInterlockStatus:=AssembleValveStatus (LowPressureInterlock:=BAV3LowPressureInterlock,
											AnotherValveOpenInterlock:=BAV3LockedBAV1Opened OR BAV3LockedBAV2Opened OR BAV3LockedSHVOpened,
											Interlock:=BAV3.xInterlock);
SHV.wInterlockStatus:=AssembleSHVLockStatus();

(*Блокировка при открытии иного клавапа*)
METHOD PUBLIC AnotherValveOpenInterlock : BOOL
VAR_INPUT

	OpenSignalValveLocker:	BOOL;
END_VAR

AnotherValveOpenInterlock:=OpenSignalValveLocker;
END_METHOD

METHOD AssembleSHVLockStatus : WORD
VAR_INPUT
END_VAR
IF THIS^.LowPressureRelaySignal  THEN
	SHV.xInterlock:=TRUE;
	SHV.wInterlockStatus:=1;
	RETURN;
ELSIF THIS^.CameraPressure>THIS^.SHVAccessPresure AND THIS^.TMPRunSignal THEN
	SHV.xInterlock:=TRUE;
	SHV.wInterlockStatus:=2;
	RETURN;
ELSE
	SHV.xInterlock:=FALSE;
	SHV.wInterlockStatus:=0;
END_IF
END_METHOD

METHOD AssembleValveStatus : WORD
VAR_INPUT
	LowPressureInterlock: BOOL;
	AnotherValveOpenInterlock:BOOL;
	Interlock:	REFERENCE TO BOOL;
END_VAR
IF NOT LowPressureInterlock AND NOT AnotherValveOpenInterlock THEN
	AssembleValveStatus:=ValveInterlockStatus.NO_LOCK;
	Interlock:=FALSE;
ELSIF LowPressureInterlock THEN
	AssembleValveStatus:=ValveInterlockStatus.LOW_PRESSURE_INTERLOCK;
	Interlock:=TRUE;
ELSIF AnotherValveOpenInterlock THEN
	AssembleValveStatus:=ValveInterlockStatus.LOCKER_VALVE_OPENED;
	Interlock:=TRUE;
END_IF
END_METHOD

METHOD PUBLIC LowPressureInterlock : BOOL;
VAR_INPUT

END_VAR

LowPressureInterlock:=THIS^.LowPressureRelaySignal;
END_METHOD

END_FUNCTION_BLOCK

// Function Blocks/Pumps/Interlock/PumpsInterlock
(*Функциональный блок  обработки всех блокировок насосв*)
FUNCTION_BLOCK PumpsInterlock
VAR_INPUT
	FVP: 						REFERENCE TO udtFVP;
	TMP: 						REFERENCE TO udtTMPDigital;
	CameraPressureHightLimitSP:	REAL;
	CameraPressure: 			REAL;
	FVPPressure:				REAL;
	BAV3Opened:					BOOL;
	BAV1Opened:					BOOL;
	BAV2Closed:					BOOL;
	CameraOpened: 				BOOL;
END_VAR
VAR_OUTPUT
END_VAR
VAR
	FVPOpenCameraLocked:	BOOL;
	TMPPressureLocked:		BOOL;
	TMPFVPTurnOffLocked:	BOOL;
END_VAR

FVPOpenCameraLocked:=AssembleFVPOpenCameraLocked(CameraOpened:=CameraOpened, ValveOpened:=BAV1Opened, BAV3Opened:=BAV3Opened);

TMPPressureLocked:=AssembleTMPPressureLocked(Pressure:=CameraPressure, PressureHightLimitSP:=CameraPressureHightLimitSP);

TMPFVPTurnOffLocked:=AssembleTMPFVPTurnOffLocked(FVPTurnON:=FVP.xTurnOn);

AssembleFVPInterlock(FVPOpenCameraLocked:=FVPOpenCameraLocked);
AssembleTMPInterlock(TMPFVPturnOfflocked:=TMPFVPTurnOffLocked, 
						TMPPressureLocked:=TMPPressureLocked,
						BAV2Closed:=BAV2Closed);

METHOD AssembleFVPInterlock : WORD
VAR_INPUT
FVPOpenCameraLocked: BOOL;
END_VAR
IF FVPOpenCameraLocked THEN
	FVP.xInterlock:=TRUE;
	FVPOpenCameraLocked:=1;
ELSE
	FVP.xInterlock:=FALSE;
	FVPOpenCameraLocked:=0;
END_IF
END_METHOD

METHOD PUBLIC AssembleFVPOpenCameraLocked : BOOL
VAR_INPUT
	CameraOpened: 	BOOL;
	ValveOpened:	BOOL;
	BAV3Opened:		BOOL;
END_VAR
IF CameraOpened AND ValveOpened THEN
	AssembleFVPOpenCameraLocked:=TRUE;
ELSIF CameraOpened AND NOT ValveOpened THEN
	AssembleFVPOpenCameraLocked:=FALSE;
ELSIF NOT CameraOpened AND BAV3Opened AND NOT BAV1Opened THEN
	AssembleFVPOpenCameraLocked:=TRUE;
ELSIF NOT CameraOpened AND NOT BAV3Opened THEN
	AssembleFVPOpenCameraLocked:=FALSE;
END_IF
END_METHOD

METHOD PUBLIC AssembleTMPFVPTurnOffLocked : BOOL
VAR_INPUT
	FVPTurnON:BOOL;
END_VAR
IF NOT FVPTurnON THEN
	AssembleTMPFVPTurnOffLocked:=TRUE;
ELSE
	AssembleTMPFVPTurnOffLocked:=FALSE;
END_IF
END_METHOD

METHOD AssembleTMPInterlock : WORD
VAR_INPUT
	TMPPressureLocked: 	BOOL;
	TMPFVPturnOfflocked: BOOL;
	BAV2Closed:			BOOL;
END_VAR
IF NOT TMPPressureLocked AND NOT TMPFVPturnOfflocked AND NOT BAV2Closed THEN
	THIS^.TMP.xInterlock:=FALSE;
	AssembleTMPInterlock:=0;
ELSIF TMPPressureLocked THEN
	THIS^.TMP.xInterlock:=TRUE;
	AssembleTMPInterlock:=1;
ELSIF TMPFVPturnOfflocked THEN
	THIS^.TMP.xInterlock:=TRUE;
	AssembleTMPInterlock:=2;
ELSIF BAV2Closed THEN
	THIS^.TMP.xInterlock:=TRUE;
END_IF
END_METHOD

METHOD PUBLIC AssembleTMPPressureLocked : BOOL
VAR_INPUT
	Pressure: REAL;
	PressureHightLimitSP: REAL;
END_VAR
IF Pressure>PressureHightLimitSP THEN
	AssembleTMPPressureLocked:=	TRUE;
ELSE
	AssembleTMPPressureLocked:= FALSE;
END_IF
END_METHOD

END_FUNCTION_BLOCK

// Function Blocks/TRM-151/Middleware/MC_ChannelView_ChannelTRM
FUNCTION_BLOCK MC_ChannelView_ChannelTRM
VAR_INPUT
	ChannelViewCount:			INT:=2;
	refChannelView_1:			POINTER TO BYTE;
	refChannelView_2:			POINTER TO BYTE;
	
	
	refChannelTRM: REFERENCE TO ARRAY[0..1] OF udtChannel;
	
	xSaveEvent:				REFERENCE TO BOOL; //событие сохранения View в TRM
	refChannelTRMSaveEvent: REFERENCE TO BOOL; //Событие для старта обмена новыми данными с ТРМ
	xLoadEvent:				REFERENCE TO BOOL;
	
END_VAR
VAR_OUTPUT
	xError:			BOOL;
	sErrorStatus:	WORD;
END_VAR
VAR
	xInit:			BOOL;
	ChannelView:	ARRAY [0..1] OF DINT;
	ChannelCounter:	INT;
END_VAR
VAR_TEMP
	ptrChannelView:	POINTER TO udtTRMChannelView;
END_VAR

IF NOT xInit THEN
	xInit:=TRUE;
	ChannelView[0]:=refChannelView_1;
	ChannelView[1]:=refChannelView_1;
END_IF
IF ChannelViewCount >2 THEN
	xError:=TRUE;
	sErrorStatus:=16#66;
	RETURN;
END_IF
xError:=FALSE;
sErrorStatus:=16#20;

IF xSaveEvent THEN
	xSaveEvent:=FALSE;
	FOR ChannelCounter:=0 TO ChannelViewCount-1 DO
		ptrChannelView:=ChannelView[ChannelCounter];
		refChannelTRM[ChannelCounter].Regulator.IntValue:=ptrChannelView^.xEnablePidRegualtor;
	END_FOR
	refChannelTRMSaveEvent:=TRUE;
END_IF

END_FUNCTION_BLOCK

// Function Blocks/TRM-151/Middleware/MC_InputView_InputTRM
FUNCTION_BLOCK MC_InputView_InputTRM
VAR_INPUT
	InputViewCount:	INT:=2;
	refInputView1:	POINTER TO BYTE;
	refInputView2:	POINTER TO BYTE;
	
	refInputsTRM:	REFERENCE TO udtInputs;
	
	xSaveEvent:		REFERENCE TO BOOL;// Cохранение данных
	xLoadevent:		REFERENCE TO BOOL;// Загрузка данных
	refInputTRMSaveEvent: REFERENCE TO BOOL;
END_VAR
VAR_OUTPUT
	xError:			BOOL;
	sErrorSatatus:	WORD;
END_VAR
VAR
	xInit:		BOOL:=FALSE;
	InputView: ARRAY[0..3] OF DINT;
	SaveCounter:	INT;
END_VAR
VAR_TEMP
	ptrInputView: POINTER TO udtTRMInputView;
END_VAR

IF NOT xinit THEN
	xInit:=TRUE;
	InputView[0]:=refInputView1;
	InputView[1]:=refInputView2;
END_IF
IF InputViewCount >2 THEN
	xError:=TRUE;
	sErrorSatatus:=16#66;
	RETURN;
END_IF
xError:=FALSE;
sErrorSatatus:=16#20;
(*Cохранение данных для отправки*)
IF xSaveEvent THEN
	xSaveEvent:=FALSE;
	FOR SaveCounter:=0 TO InputViewCount-1  DO
		ptrInputView:=InputView[SaveCounter];
		refInputsTRM.Input[SaveCounter].SensoreType.IntValue:=ptrInputView^.SensoreType;
		refInputsTRM.Input[SaveCounter].DigitalFiltertimeConstant.IntValue:=ptrInputView^.DigitalFiltertimeConst;
		refInputsTRM.Input[SaveCounter].DigitalFilterline.IntValue:=ptrInputView^.DigitalFilterLine;
		refInputsTRM.Input[SaveCounter].PollingSensoreTime.FloatValue:=ptrInputView^.PollingSensoreTime;
		refInputsTRM.Input[SaveCounter].LowEdgeSensoreChange.IntValue:=ptrInputView^.LowEdgeSensoreChange;
		refInputsTRM.Input[SaveCounter].HightEdgeSensoreChange.IntValue:=ptrInputView^.HightEdgeSensoreChange;
		refInputsTRM.Input[SaveCounter].CorrectionOfShiftCharacteristic.IntValue:=ptrInputView^.CorrectionOfCharacteresticShift;
		refInputsTRM.Input[SaveCounter].CorrectionOfInclineCharacterisitc.FloatValue:=ptrInputView^.CorrectionOfInclineCharacteristic;
	END_FOR
	refInputTRMSaveEvent:=TRUE;
END_IF
(*Извлечение данных после загрузки*)
IF xLoadEvent THEN
	xLoadEvent:=FALSE;
	FOR SaveCounter:=0 TO InputViewCount-1  DO
		ptrInputView:=InputView[SaveCounter];
		ptrInputView^.DigitalFiltertimeConst:=refInputsTRM.Input[SaveCounter].DigitalFiltertimeConstant.IntValue;
		ptrInputView^.DigitalFilterLine:=refInputsTRM.Input[SaveCounter].DigitalFilterline.IntValue;
		ptrInputView^.PollingSensoreTime:=refInputsTRM.Input[SaveCounter].PollingSensoreTime.FloatValue;
		ptrInputView^.LowEdgeSensoreChange:=refInputsTRM.Input[SaveCounter].LowEdgeSensoreChange.IntValue;
		ptrInputView^.HightEdgeSensoreChange:=refInputsTRM.Input[SaveCounter].HightEdgeSensoreChange.IntValue;
		ptrInputView^.CorrectionOfCharacteresticShift:=refInputsTRM.Input[SaveCounter].CorrectionOfShiftCharacteristic.IntValue;
		ptrInputView^.CorrectionOfInclineCharacteristic:=refInputsTRM.Input[SaveCounter].CorrectionOfInclineCharacterisitc.FloatValue;
	END_FOR
END_IF

END_FUNCTION_BLOCK

// Function Blocks/TRM-151/Middleware/MC_OperatingView_OperatingTRM
FUNCTION_BLOCK MC_OperatingView_OperatingTRM
VAR_INPUT
	refOperationParametr:	REFERENCE TO udtOperationParameters;
	refOperationView:		POINTER TO udtTRMOperatingView;
	StartCommand:			REFERENCE TO TRMStartSignal;
	xSaveEvent:				REFERENCE TO BOOL; 
	xReadEvent:				REFERENCE TO BOOL; //Чтение данных с ТРМ
	xStartStopEvent:		REFERENCE TO BOOL;
END_VAR
VAR_OUTPUT
END_VAR
VAR
	xInit:				BOOL;
	PowerFeedback:		ARRAY [0..1] OF  DINT;
	PowerFeedbackUnit:	POINTER TO REAL;
	ReadFeedback:		ARRAY[0..1] OF  DINT;
	ReadFeedbackUnit:	POINTER TO REAL;
	Readcounter:INT;
END_VAR

IF NOT xInit THEN
	xInit:=TRUE;
	PowerFeedback[0]:=	 ADR(refOperationView^.rPowerFeedbackChannel_1);
	PowerFeedback[1]:=	 ADR(refOperationView^.rPowerFeedbackChannel_2);
	ReadFeedback[0]:=	ADR(refOperationView^.rReadfeedbackChannel_1);
	ReadFeedback[1]:=	ADR(refOperationView^.rReadfeedbackChannel_1);
END_IF

IF xSaveEvent THEN
	xSaveEvent:=FALSE;
	refOperationParametr.ProgramNumberFeedback.IntValue:=refOperationView^.ProgrammNoSP-1;
	refOperationParametr.StepNumberFeedback.IntValue:=refOperationView^.ProgramStepNoSP-1;
END_IF

IF xStartStopEvent THEN
	xStartStopEvent:=FALSE;
	refOperationParametr.StarCommand.IntValue:=refOperationView^.StartProcessSignal;
END_IF
//Вычитка данных во время цикла работы.
IF xReadEvent THEN
	xReadEvent:=FALSE;
	refOperationView^.ProgramNoFb:=refOperationParametr.ProgramNumberFeedback.IntValue;
	refOperationView^.ProgramStepNoFb:=refOperationParametr.StepNumberFeedback.IntValue;
	FOR Readcounter:=0 TO 1 DO
		PowerFeedbackUnit:=PowerFeedback[Readcounter];
		ReadFeedbackUnit:=ReadFeedback[Readcounter];
		PowerFeedbackUnit^:=refOperationParametr.PowerFeedback[Readcounter].Value.FloatValue;
		ReadFeedbackUnit^:=refOperationParametr.RegulatorSetPointfeedback[Readcounter].Value.FloatValue;
	END_FOR
END_IF

END_FUNCTION_BLOCK

// Function Blocks/TRM-151/Middleware/MC_OutputView_OutputTRM
FUNCTION_BLOCK MC_OutputView_OutputTRM
VAR_INPUT
	OutputViewCount:		INT:=2;
	refOutputView_1:		POINTER TO BYTE;
	refOutputView_2:		POINTER TO BYTE;
	
	refOutputTRM:			REFERENCE TO udtSignalConverters;
	
	xSaveEvent:				REFERENCE TO BOOL;
	xLoadEvent:				REFERENCE TO BOOL;
	refOutputTRMSaveEvent:	REFERENCE TO BOOL;
END_VAR
VAR_OUTPUT
	xError:			BOOL;
	sErrorStatus:	WORD;
END_VAR
VAR
	xInit:		BOOL;
	OutputView:	ARRAY [0..1] OF DINT;
	SaveCounter:INT;
END_VAR
VAR_TEMP
	ptrOutputView:	POINTER TO udtTRMOutput;
END_VAR

IF NOT xInit THEN
	xInit:=TRUE;
	OutputView[0]:=refOutputView_1;
	OutputView[1]:=refOutputView_2;
END_IF
IF OutputViewCount >2 THEN
	xError:=TRUE;
	sErrorStatus:=16#66;
	RETURN;
END_IF
xError:=FALSE;
sErrorStatus:=16#20;
IF xSaveEvent THEN
	xSaveEvent:=FALSE;
	FOR SaveCounter:=0 TO OutputViewCount-1 DO
		ptrOutputView:=OutputView[SaveCounter];
		refOutputTRM.SignalConverter[SaveCounter].MaxOutputPower.FloatValue:=ptrOutputView^.MaxOutputPower;
		refOutputTRM.SignalConverter[SaveCounter].MaxSpeedOutputPowerSpeed.FloatValue:=ptrOutputView^.MaxSpeedOutputPowerSpeed;
		refOutputTRM.SignalConverter[SaveCounter].MinOutputPower.FloatValue:=ptrOutputView^.MinOutputPower;
	END_FOR
	refOutputTRMSaveEvent:=TRUE;
END_IF

END_FUNCTION_BLOCK

// Function Blocks/TRM-151/Middleware/MC_ProgramOfTecholog_ProgramOfTechnologTRM
FUNCTION_BLOCK MC_ProgramOfTecholog_ProgramOfTechnologTRM
VAR_INPUT
	refTechnologView:		REFERENCE TO udtTRMTechnologOperation;
	refTechonologTRM:		REFERENCE TO udtProgramOfTechnolog;
	refStepSetpoint:		REFERENCE TO udtSetPoints;
	refProgramOfTechnologSaveEvent:	REFERENCE To BOOL;
END_VAR
VAR_OUTPUT
END_VAR
VAR
	SaveCountProgram:				INT;
	SaveCountStep:					INT;
END_VAR

IF refTechnologView.xSaveEvent THEN
	refTechnologView.xSaveEvent:=FALSE;
	refTechonologTRM.StartProgramSource.IntValue:=refTechnologView.StartProgramSource;
	refTechonologTRM.TimeScaleInProgram.IntValue:=refTechnologView.TimeFormat;
	FOR SaveCountProgram:=0 TO 11 DO
		refTechonologTRM.Programs[SaveCountProgram].ProgramNumber:=SaveCountProgram*10;
		refTechonologTRM.Programs[SaveCountProgram].StarProgrammAccept.IntValue:=refTechnologView.TechnologOperationProgram[SaveCountProgram].StartProgramPermit;
		FOR SaveCountStep:=0 TO 10 DO
			refTechonologTRM.Programs[SaveCountProgram].Steps[SaveCountStep].StepId:=SaveCountStep+SaveCountProgram*10;
			refTechonologTRM.Programs[SaveCountProgram].Steps[SaveCountStep].StepType.IntValue:=refTechnologView.TechnologOperationProgram[SaveCountProgram].Step[SaveCountStep].StepType;
			refTechonologTRM.Programs[SaveCountProgram].Steps[SaveCountStep].ProgramNumberToTransition.IntValue:=refTechnologView.TechnologOperationProgram[SaveCountProgram].Step[SaveCountStep].TransactionProgramNo;
			refTechonologTRM.Programs[SaveCountProgram].Steps[SaveCountStep].StepNumberToTransition.IntValue:=refTechnologView.TechnologOperationProgram[SaveCountProgram].Step[SaveCountStep].TransactionStepNo;
			refTechonologTRM.Programs[SaveCountProgram].Steps[SaveCountStep].NextStepTransitionLogic.IntValue:=refTechnologView.TechnologOperationProgram[SaveCountProgram].Step[SaveCountStep].NextSteptransactionLogic;
			refTechonologTRM.Programs[SaveCountProgram].Steps[SaveCountStep].SPTransitionCondition.IntValue:=refTechnologView.TechnologOperationProgram[SaveCountProgram].Step[SaveCountStep].TransactionConditionValue;
			refTechonologTRM.Programs[SaveCountProgram].Steps[SaveCountStep].ComputeNumberValueSourceToTrasition.IntValue:=refTechnologView.TechnologOperationProgram[SaveCountProgram].Step[SaveCountStep].InputNumberTransactionValue;
			refTechonologTRM.Programs[SaveCountProgram].Steps[SaveCountStep].SPValueToTransition.FloatValue:= refTechnologView.TechnologOperationProgram[SaveCountProgram].Step[SaveCountStep].SetPoint;
			refTechonologTRM.Programs[SaveCountProgram].Steps[SaveCountStep].StepTime.FloatValue:=refTechnologView.TechnologOperationProgram[SaveCountProgram].Step[SaveCountStep].StepLatency;
			refStepSetpoint.Programs[SaveCountProgram].Steps[SaveCountStep].SetpointID:=SavecountStep+SaveCountProgram*10;
			refStepSetpoint.Programs[SaveCountProgram].Steps[SaveCountStep].SetPointType.IntValue:=refTechnologView.TechnologOperationProgram[SaveCountProgram].StepSetPoint[SaveCountStep].SetPointType;
			refStepSetpoint.Programs[SaveCountProgram].Steps[SaveCountStep].SetPointSpeed.FloatValue:=refTechnologView.TechnologOperationProgram[SaveCountProgram].StepSetPoint[SaveCountStep].SetpointSpeed;
			refStepSetpoint.Programs[SaveCountProgram].Steps[SaveCountStep].MinSetPoint.FloatValue:=refTechnologView.TechnologOperationProgram[SaveCountProgram].StepSetPoint[SaveCountStep].MinSetpoint;
			refStepSetpoint.Programs[SaveCountProgram].Steps[SaveCountStep].MaxSetPoint.FloatValue:=refTechnologView.TechnologOperationProgram[SaveCountProgram].StepSetPoint[SaveCountStep].MaxSetpoint;
		END_FOR
	END_FOR
	refProgramOfTechnologSaveEvent:=TRUE;
END_IF

END_FUNCTION_BLOCK

// Function Blocks/TRM-151/Middleware/MC_RegulatorView_RegulatorTRM
FUNCTION_BLOCK MC_RegulatorView_RegulatorTRM
VAR_INPUT
	RegulatorViewCount:		INT:=2;
	refRegulatorView_1:		POINTER TO BYTE;
	refRegulatorView_2:		POINTER TO BYTE;
	
	
	refRegulatorsTRM:		REFERENCE TO udtRegulators;
	
	xSaveEvent:				REFERENCE TO BOOL;
	xLoadEvent:				REFERENCE TO BOOL;
	
END_VAR
VAR_OUTPUT
	xError:			BOOL;
	sErrorStatus:	WORD;
END_VAR
VAR
	xInit:			BOOL;
	RegulatorView:	ARRAY[0..1] OF DINT;
	RegulatorCounter:	INT;
END_VAR
VAR_TEMP
	ptrRegulatorView:	POINTER TO udtTRMRegulatorView;
END_VAR

IF NOT xInit THEN
	xInit:=TRUE;
	RegulatorView[0]:=refRegulatorView_1;
	RegulatorView[1]:=refRegulatorView_2;
END_IF
IF RegulatorViewCount >2 THEN
	xError:=TRUE;
	sErrorStatus:=16#66;
	RETURN;
END_IF
xError:=FALSE;
sErrorStatus:=16#20;
IF xSaveEvent THEN
	xSaveEvent:=FALSE;
	FOR RegulatorCounter:=0 TO RegulatorViewCount-1 DO
		ptrRegulatorView:=RegulatorView[RegulatorCounter];
		refRegulatorsTRM.Regulator[RegulatorCounter].Deadband.FloatValue:=ptrRegulatorView^.Deadband;
		refRegulatorsTRM.Regulator[RegulatorCounter].RegulatorMode.IntValue:=ptrRegulatorView^.RegulationMode;
		refRegulatorsTRM.Regulator[RegulatorCounter].PIDRegulator.PCoeff.FloatValue:=ptrRegulatorView^.PIDRegualtor.PCoeff;
		refRegulatorsTRM.Regulator[RegulatorCounter].PIDRegulator.ICoeff.FloatValue:=ptrRegulatorView^.PIDRegualtor.ICoeff;//TODO: посмотреть конвертацию MGU-25
		refRegulatorsTRM.Regulator[RegulatorCounter].PIDRegulator.DIDifF.FloatValue:=ptrRegulatorView^.PIDRegualtor.DIDiff;
		refRegulatorsTRM.Regulator[RegulatorCounter].PIDRegulator.NominalPower.FloatValue:=ptrRegulatorView^.PIDRegualtor.NominalPower;
		refRegulatorsTRM.Regulator[RegulatorCounter].PIDRegulator.MaxIntegralLimit.FloatValue:=ptrRegulatorView^.PIDRegualtor.MaxIntegralLimit;
		refRegulatorsTRM.Regulator[RegulatorCounter].PIDRegulator.MinIntegralLimit.FloatValue:=ptrRegulatorView^.PIDRegualtor.MinIntegralLimit;
	END_FOR
END_IF

END_FUNCTION_BLOCK

// Function Blocks/TRM-151/Pooling/MC_TRMPooling
(*Deprecate*)
FUNCTION_BLOCK MC_TRMPooling
VAR_INPUT
	refChannelTRMSaveEvent: 			REFERENCE TO BOOL;
	refOutputTRMSaveEvent:				REFERENCE TO BOOL;
	refInputTRMSaveEvent:				REFERENCE TO BOOL;
	refprogramOfTechnologTRMSaveEvent: 	REFERENCE TO BOOL;
	refOperatingTRMSaveEvent: 			REFERENCE TO BOOL;
	refOperatingTRMLoadEvent: 			REFERENCE TO BOOL;
	refOperatingTRMStartStopEvent: 		REFERENCE TO BOOL;
	xAcknowledgment:					REFERENCE TO BOOL; //Cигнал о сбросе ошибки FB;
	
	
	ptrChannelsTRM:						POINTER TO ARRAY[0..1] OF udtChannel;
	ptrInputsTRM:						POINTER TO udtInputs;
	ptrOutputTRM:						POINTER TO udtSignalConverters;
	ptrProgramOfTechnologTRM: 			POINTER TO udtProgramOfTechnolog;
	ptrProgramOfTechnologSetpoint: 		POINTER TO udtSetPoints;
	ptrOperatingParametrTRM: 			POINTER TO udtOperationParameters;
END_VAR
VAR_OUTPUT
	xTRMPoolingError:BOOL; //Общая ошибка пулинга
	xTRMWriteError: BOOL;
	xTRMReadError:	BOOL;
	wTRMWriteError: WORD;
	wTRMReadError:	WORD;
END_VAR
VAR
	FIFO: 					FIFO.FIFO;
	WriteInt: 				OwenNet.OWEN_SET_DINT;
	WriteFloat: 			OwenNet.OWEN_SET_REAL;
	ReadWriteOther: 		OwenNet.OWEN_UNI_IO;
	ReadInt: 				OwenNet.OWEN_GET_DINT;
	ReadFloat: 				OwenNet.OWEN_GET_REAL;
	iStage: 				INT:=TRM_POOLING_STAGE.WAIT;
	iChannelTRMCount: 		INT;
	iStructElement:			INT;
	ptrChannelTRM:			POINTER TO BYTE;
	xOperationStage:		BOOL;
	xPushError:				BOOL;//Ошибка добавления в очередь
	iPopError:				INT;
	xInit:					BOOL:=FALSE;
	xSenderError:			BOOL;
	wSenderError:			WORD;
	xSenderComplete:		BOOL;
	xReaderError:			BOOL;
	wReaderError:			WORD;
	xReaderComplete:		BOOL;
	iStageErrorCallback: 	INT; //Стадия выхода в ошибку
	xFBError:				BOOL;
END_VAR
VAR RETAIN
	iErrorCount: INT;
END_VAR

IF NOT xInit THEN
	(*Реализация инициализайции FB OwenNet*)
	xInit:=TRUE;
END_IF
IF xAcknowledgment THEN
	xAcknowledgment:=FALSE;
	xFBError:=FALSE;
	iErrorCount:=0;
END_IF
CASE iStage OF
	TRM_POOLING_STAGE.WAIT:
		IF xFBError THEN
			RETURN;
		END_IF
		//действия при полной очереди
		IF FIFO.isFull THEN
			iStage:=TRM_POOLING_STAGE.GET_ACTION;
			RETURN;
		END_IF
		//действия при стадии опроса
		IF xOperationStage THEN
			IF FIFO.isEmpty THEN
				xOperationStage:=FALSE;
				RETURN;
			END_IF
			iStage:=TRM_POOLING_STAGE.GET_ACTION;
			RETURN;	
		END_IF
		//Заполенение очереди на опрос
		IF refChannelTRMSaveEvent THEN
			F_TRMAddEventHandler(refFIFO:= ADR(FIFO),
				Stage:=TRM_POOLING_STAGE.ChanellTRM_SAVE,
				refEvent:=ADR(refChannelTRMSaveEvent),
				xError=>xPushError);
			IF xPushError THEN
				RETURN;
			END_IF
		END_IF
		
		IF refInputTRMSaveEvent THEN
				F_TRMAddEventHandler(refFIFO:= ADR(FIFO),
				Stage:=TRM_POOLING_STAGE.InputTRM_SAVE,
				refEvent:=ADR(refInputTRMSaveEvent),
				xError=>xPushError);
			IF xPushError THEN
				RETURN;
			END_IF
		END_IF
		
		IF refOutputTRMSaveEvent THEN
			F_TRMAddEventHandler(refFIFO:= ADR(FIFO),
				Stage:=TRM_POOLING_STAGE.OutputTRM_SAVE,
				refEvent:=ADR(refOutputTRMSaveEvent),
				xError=>xPushError);
			IF xPushError THEN
				RETURN;
			END_IF
		END_IF
		
		IF refProgramOfTechnologTRMSaveEvent THEN
				F_TRMAddEventHandler(refFIFO:= ADR(FIFO),
				Stage:=TRM_POOLING_STAGE.ProgramOfTechonologTRM_SAVE,
				refEvent:=ADR(refProgramOfTechnologTRMSaveEvent),
				xError=>xPushError);
			IF xPushError THEN
				RETURN;
			END_IF
		END_IF
		
		IF refOperatingTRMSaveEvent THEN
				F_TRMAddEventHandler(refFIFO:= ADR(FIFO),
				Stage:=TRM_POOLING_STAGE.OperatingTRM_SAVE,
				refEvent:=ADR(refOperatingTRMSaveEvent),
				xError=>xPushError);
			IF xPushError THEN
				RETURN;
			END_IF
		END_IF
		
		IF refOperatingTRMStartStopEvent THEN
				F_TRMAddEventHandler(refFIFO:= ADR(FIFO),
				Stage:=TRM_POOLING_STAGE.OperatingTRM_STARTSTOP,
				refEvent:=ADR(refOperatingTRMStartStopEvent),
				xError=>xPushError);
			IF xPushError THEN
				RETURN;
			END_IF
		END_IF
		F_TRMAddEventHandler(refFIFO:= ADR(FIFO),
				Stage:=TRM_POOLING_STAGE.OperatingTRM_LOAD,
				refEvent:=ADR(refOperatingTRMLoadEvent),
				xError=>xPushError);
		IF xPushError THEN
				RETURN;
		END_IF
		TRM_POOLING_STAGE.GET_ACTION:
			IF FIFO.isEmpty THEN
				iStage:=TRM_POOLING_STAGE.WAIT;
				RETURN;
			END_IF
			iStage:=FIFO.Pop(ptrErr:=ADR(iPopError));
			IF iPopError = FIFO.FIFO_ERR.NO_ERROR THEN
				RETURN;
			END_IF
			iStage:=TRM_POOLING_STAGE.WAIT;
			
		(*____________________________*)	
		TRM_POOLING_STAGE.ChanellTRM_SAVE:
			F_TRMSender(ptrStruct:=ptrChannelsTRM,
						uiStructureSize:=SIZEOF(ptrChannelTRM^),
						uiSize:=SIZEOF(ptrChannelTRM^)/SIZEOF(OwenValue),
						ptrWriteFloat :=ADR(WriteFloat),
						ptrWriteInt := ADR(WriteInt),
						ptrWriteOther := ADR(ReadWriteOther),
						xError=>xSenderError,
						Error=>wSenderError,
						Complete=>xSenderComplete);
			IF xSenderComplete THEN
				iStage:=TRM_POOLING_STAGE.WAIT;
				xSenderComplete:=FALSE;
				RETURN;
			END_IF
			IF xSenderError THEN
				iStageErrorCallback:=iStage;
				iStage:=TRM_POOLING_STAGE.ERROR;
				RETURN;
			END_IF
			
			(*--------------------------------------*)
			TRM_POOLING_STAGE.InputTRM_SAVE:
				F_TRMSender(
						ptrStruct:=ptrInputsTRM,
						uiStructureSize:=SIZEOF(udtInputs),
						uiSize:=SIZEOF(udtInputs)/SIZEOF(OwenValue),
						ptrWriteFloat :=ADR(WriteFloat),
						ptrWriteInt := ADR(WriteInt),
						ptrWriteOther := ADR(ReadWriteOther),
						xError=>xSenderError,
						Error=>wSenderError,
						Complete=>xSenderComplete);
				IF xSenderComplete THEN
					iStage:=TRM_POOLING_STAGE.WAIT;
					xSenderComplete:=FALSE;
					RETURN;
				END_IF
				IF xSenderError THEN
					iStageErrorCallback:=iStage;
					iStage:=TRM_POOLING_STAGE.ERROR;
					RETURN;
				END_IF
			TRM_POOLING_STAGE.OutputTRM_SAVE:
				F_TRMSender(
						ptrStruct:=ptrOutputTRM,
						uiStructureSize:=SIZEOF(udtSignalConverters),
						uiSize:=SIZEOF(udtSignalConverters)/SIZEOF(OwenValue),
						ptrWriteFloat :=ADR(WriteFloat),
						ptrWriteInt := ADR(WriteInt),
						ptrWriteOther := ADR(ReadWriteOther),
						xError=>xSenderError,
						Error=>wSenderError,
						Complete=>xSenderComplete);
				IF xSenderComplete THEN
					iStage:=TRM_POOLING_STAGE.WAIT;
					xSenderComplete:=FALSE;
					RETURN;
				END_IF
				IF xSenderError THEN
					iStageErrorCallback:=iStage;
					iStage:=TRM_POOLING_STAGE.ERROR;
					RETURN;
				END_IF
			TRM_POOLING_STAGE.ProgramOfTechonologTRM_SAVE:
				F_TRMSender(
						ptrStruct:=ptrProgramOfTechnologTRM,
						uiStructureSize:=SIZEOF(udtProgramOfTechnolog),
						uiSize:=SIZEOF(udtProgramOfTechnolog)/SIZEOF(OwenValue),
						ptrWriteFloat :=ADR(WriteFloat),
						ptrWriteInt := ADR(WriteInt),
						ptrWriteOther := ADR(ReadWriteOther),
						xError=>xSenderError,
						Error=>wSenderError,
						Complete=>xSenderComplete);
				IF xSenderComplete THEN
					iStage:=TRM_POOLING_STAGE.ProgramOfTechonologTRM_SETPOINT_SAVE;
					xSenderComplete:=FALSE;
					RETURN;
				END_IF
				IF xSenderError THEN
					iStageErrorCallback:=iStage;
					iStage:=TRM_POOLING_STAGE.ERROR;
					RETURN;
				END_IF
			TRM_POOLING_STAGE.ProgramOfTechonologTRM_SETPOINT_SAVE:
				F_TRMSender(
						ptrStruct:=ptrProgramOfTechnologSetpoint,
						uiStructureSize:=SIZEOF(udtSetPoints),
						uiSize:=SIZEOF(udtSetPoints)/SIZEOF(OwenValue),
						ptrWriteFloat :=ADR(WriteFloat),
						ptrWriteInt := ADR(WriteInt),
						ptrWriteOther := ADR(ReadWriteOther),
						xError=>xSenderError,
						Error=>wSenderError,
						Complete=>xSenderComplete);
				IF xSenderComplete THEN
					iStage:=TRM_POOLING_STAGE.WAIT;
					xSenderComplete:=FALSE;
					RETURN;
				END_IF
				IF xSenderError THEN
					iStageErrorCallback:=iStage;
					iStage:=TRM_POOLING_STAGE.ERROR;
					RETURN;
				END_IF
			TRM_POOLING_STAGE.OperatingTRM_STARTSTOP:
				F_TRMSender(
						ptrStruct:=ptrOperatingParametrTRM,
						uiStructureSize:=SIZEOF(udtOperationParameters),
						uiSize:=1,
						ptrWriteFloat :=ADR(WriteFloat),
						ptrWriteInt := ADR(WriteInt),
						ptrWriteOther := ADR(ReadWriteOther),
						xError=>xSenderError,
						Error=>wSenderError,
						Complete=>xSenderComplete);
				IF xSenderComplete THEN
					iStage:=TRM_POOLING_STAGE.WAIT;
					xSenderComplete:=FALSE;
					RETURN;
				END_IF
				IF xSenderError THEN
					iStageErrorCallback:=iStage;
					iStage:=TRM_POOLING_STAGE.ERROR;
					RETURN;
				END_IF
			TRM_POOLING_STAGE.OperatingTRM_SAVE:
					F_TRMSender(
						ptrStruct:=ptrOperatingParametrTRM+2*SIZEOF(OwenValue),
						uiStructureSize:=SIZEOF(udtOperationParameters),
						uiSize:=2,
						ptrWriteFloat :=ADR(WriteFloat),
						ptrWriteInt := ADR(WriteInt),
						ptrWriteOther := ADR(ReadWriteOther),
						xError=>xSenderError,
						Error=>wSenderError,
						Complete=>xSenderComplete);
				IF xSenderComplete THEN
					iStage:=TRM_POOLING_STAGE.WAIT;
					xSenderComplete:=FALSE;
					RETURN;
				END_IF
				IF xSenderError THEN
					iStageErrorCallback:=iStage;
					iStage:=TRM_POOLING_STAGE.ERROR;
					RETURN;
				END_IF
			TRM_POOLING_STAGE.OperatingTRM_LOAD:
					F_TRMReader(
						ptrStruct:=	ptrOperatingParametrTRM,
						uiStructureSize:=SIZEOF(udtOperationParameters),
						uiSize:=SIZEOF(udtOperationParameters)/SIZEOF(OwenValue),
						ptrReadInt:=ADR(ReadInt),
						ptrReadFloat:=ADR(ReadFloat),
						ptrReadOther:=ADR(ReadWriteOther),
						xError=>xReaderError,
						Error=>wReaderError,
						Complete=>xReaderComplete);
					IF xReaderComplete THEN
						refOperatingTRMLoadEvent:=TRUE;
						iStage:=TRM_POOLING_STAGE.WAIT;
						xReaderComplete:=FALSE;
						RETURN;
					END_IF
					IF xReaderError THEN
						iStageErrorCallback:=iStage;
						iStage:=TRM_POOLING_STAGE.ERROR;
						RETURN;
					END_IF
			TRM_POOLING_STAGE.ERROR:
				iErrorCount:=iErrorCount+1;
				IF iErrorCount > 5 THEN
					xFBError:=TRUE;
				END_IF
				iStage:=TRM_POOLING_STAGE.WAIT;
				IF iStageErrorCallback = TRM_POOLING_STAGE.InputTRM_SAVE THEN
					refInputTRMSaveEvent:=TRUE;
				END_IF
				IF iStageErrorCallback = TRM_POOLING_STAGE.OutputTRM_SAVE THEN
					refOperatingTRMSaveEvent:=TRUE;
				END_IF
				IF iStageErrorCallback = TRM_POOLING_STAGE.ProgramOfTechonologTRM_SAVE THEN
					refprogramOfTechnologTRMSaveEvent:=TRUE;
				END_IF
				IF iStageErrorCallback = TRM_POOLING_STAGE.ProgramOfTechonologTRM_SETPOINT_SAVE THEN
					refprogramOfTechnologTRMSaveEvent:=TRUE;
				END_IF
				IF iStageErrorCallback = TRM_POOLING_STAGE.OperatingTRM_SAVE THEN
					refOperatingTRMSaveEvent:=TRUE;
				END_IF
				IF iStageErrorCallback = TRM_POOLING_STAGE.OperatingTRM_STARTSTOP THEN
					refOperatingTRMStartStopEvent:=TRUE;
				END_IF
				IF iStageErrorCallback = TRM_POOLING_STAGE.ChanellTRM_SAVE THEN
					refChannelTRMSaveEvent:=TRUE;
				END_IF
				IF iStageErrorCallback = TRM_POOLING_STAGE.OperatingTRM_LOAD THEN
					refOperatingTRMLoadEvent:=TRUE;
				END_IF
				iStageErrorCallback:=0;
				Return;	
						
END_CASE	
xTRMPoolingError:= xFBError;
xTRMWriteError:=xSenderError;
xTRMReadError:=xReaderError;
wTRMWriteError:=wSenderError;
wTRMReadError:=wReaderError;

END_FUNCTION_BLOCK

// Function Blocks/VacuumCamera/Pumping/VacuumCameraWithoutSHV
FUNCTION_BLOCK VacuumCameraWithoutSHV
VAR_INPUT
	xStartVacuumProcessOperatorCommand:		REFERENCE TO BOOL; //Командна на старт процкесса откачки
	xStartDevacuumProcessOperatorCommand:	REFERENCE TO BOOL; //Команда на старт процесса напуска воздуха
	xStopVacuumProcesOoperatorCommand:		REFERENCE TO BOOL; //Команада на остановку работы вакуумной камеры
	xStopAnyProcessCommandFromOperator:		REFERENCE TO BOOL; //Команда на остановку любого процесса от оператора.
	xProcessResumeCommand:					REFERENCE TO BOOL;	//Команда продолжения процесса откачки с момента вознкиновения ошибки
	xProcessAbort:							REFERENCE TO BOOL;  //Команда сброса процесса откачки в начальное положение при ошибке
	BAV1:									REFERENCE TO udtValve;
	BAV1Setting:							REFERENCE TO udtValveSetting;
	BAV2:									REFERENCE TO udtValve;
	BAV2Setting:							REFERENCE TO udtValveSetting;
	BAV3:									REFERENCE TO udtValve;
	BAV3Setting:							REFERENCE TO udtValveSetting;
	TMP:									REFERENCE TO udtTMPDigital;
	TMPSetting:								REFERENCE TO udtTMPDigitalSetting;
	FVP:									REFERENCE TO udtFVP;
	FVPSetting:								REFERENCE TO udtFVPSetting;
	VacuumCamera:							REFERENCE TO udtVacuumCamera;
	VacuumCameraSetting:					REFERENCE TO udtVacuumCameraSetting;
	ClosedCameraSensore:					REFERENCE TO udtDiscreteSignal;
	TMPBreakingValve:						REFERENCE TO udtValve;
	TMPBreakingValveSetting:				REFERENCE TO udtValveSetting;
	CameraPressure:							REFERENCE TO udtPressureSensore;
	FVPPressure:							REFERENCE TO udtPressureSensore;
	
END_VAR
VAR_OUTPUT
	wError: 	WORD;
	Status: 	WORD;
	xError: 	BOOL;

